LIN {X 0.039,Y -218.237,Z 1468.192,A 0.000,B 0.000,C 90.000,E1 34.612} C_DIS
LIN {X 0.042,Y -211.829,Z 1468.171,A 0.000,B 0.000,C 90.000,E1 30.718} C_DIS
LIN {X -0.038,Y -206.290,Z 1468.149,A 0.000,B 0.000,C 90.000,E1 26.796} C_DIS
LIN {X 0.085,Y -201.468,Z 1468.127,A 0.000,B 0.000,C 90.000,E1 22.770} C_DIS
LIN {X 0.019,Y -196.661,Z 1468.100,A 0.000,B 0.000,C 90.000,E1 17.946} C_DIS
LIN {X -0.013,Y -192.947,Z 1468.073,A 0.000,B 0.000,C 90.000,E1 13.063} C_DIS
LIN {X 0.033,Y -189.936,Z 1468.041,A 0.000,B 0.000,C 90.000,E1 7.296} C_DIS
LIN {X 0.003,Y -188.141,Z 1468.004,A 0.000,B 0.000,C 90.000,E1 0.688} C_DIS
LIN {X -0.094,Y -187.890,Z 1467.974,A 0.000,B 0.000,C 90.000,E1 355.412} C_DIS
LIN {X -0.024,Y -189.029,Z 1467.938,A 0.000,B 0.000,C 90.000,E1 348.757} C_DIS
LIN {X 0.018,Y -191.542,Z 1467.905,A 0.000,B 0.000,C 90.000,E1 342.960} C_DIS
LIN {X 0.031,Y -194.968,Z 1467.878,A 0.000,B 0.000,C 90.000,E1 338.028} C_DIS
LIN {X 0.048,Y -198.751,Z 1467.855,A 0.000,B 0.000,C 90.000,E1 333.948} C_DIS
LIN {X 0.000,Y -203.644,Z 1467.833,A 0.000,B 0.000,C 90.000,E1 329.921} C_DIS
LIN {X 0.050,Y -208.477,Z 1467.815,A 0.000,B 0.000,C 90.000,E1 326.707} C_DIS
LIN {X 0.045,Y -214.140,Z 1467.797,A 0.000,B 0.000,C 90.000,E1 323.543} C_DIS
LIN {X -0.033,Y -220.739,Z 1467.780,A 0.000,B 0.000,C 90.000,E1 320.436} C_DIS
LIN {X -0.092,Y -229.220,Z 1467.761,A 0.000,B 0.000,C 90.000,E1 316.986} C_DIS
LIN {X 0.104,Y -238.990,Z 1467.742,A 0.000,B 0.000,C 90.000,E1 313.542} C_DIS
LIN {X -0.060,Y -248.706,Z 1467.726,A 0.000,B 0.000,C 90.000,E1 310.620} C_DIS
LIN {X 0.027,Y -256.867,Z 1467.714,A 0.000,B 0.000,C 90.000,E1 308.418} C_DIS
LIN {X -0.032,Y -267.355,Z 1467.700,A 0.000,B 0.000,C 90.000,E1 305.931} C_DIS
LIN {X -0.147,Y -275.740,Z 1467.690,A 0.000,B 0.000,C 90.000,E1 304.199} C_DIS
LIN {X 0.156,Y -283.214,Z 1467.682,A 0.000,B 0.000,C 90.000,E1 302.752} C_DIS
LIN {X -0.016,Y -295.382,Z 1467.671,A 0.000,B 0.000,C 90.000,E1 300.747} C_DIS
LIN {X -0.006,Y -304.284,Z 1467.663,A 0.000,B 0.000,C 90.000,E1 299.411} C_DIS
LIN {X -0.072,Y -311.630,Z 1467.658,A 0.000,B 0.000,C 90.000,E1 298.437} C_DIS
LIN {X 0.129,Y -322.365,Z 1467.651,A 0.000,B 0.000,C 90.000,E1 297.129} C_DIS
LIN {X -0.024,Y -344.394,Z 1467.638,A 0.000,B 0.000,C 90.000,E1 294.823} C_DIS
LIN {X -0.093,Y -358.123,Z 1467.630,A 0.000,B 0.000,C 90.000,E1 293.462} C_DIS
LIN {X 0.175,Y -368.842,Z 1467.624,A 0.000,B 0.000,C 90.000,E1 292.333} C_DIS
LIN {X -0.167,Y -379.420,Z 1467.618,A 0.000,B 0.000,C 90.000,E1 291.280} C_DIS
LIN {X -0.060,Y -392.204,Z 1467.610,A 0.000,B 0.000,C 90.000,E1 289.885} C_DIS
LIN {X -0.036,Y -402.044,Z 1467.604,A 0.000,B 0.000,C 90.000,E1 288.779} C_DIS
LIN {X 0.133,Y -411.649,Z 1467.598,A 0.000,B 0.000,C 90.000,E1 287.638} C_DIS
LIN {X -0.221,Y -418.371,Z 1467.594,A 0.000,B 0.000,C 90.000,E1 286.858} C_DIS
LIN {X -0.109,Y -424.471,Z 1467.589,A 0.000,B 0.000,C 90.000,E1 286.024} C_DIS
LIN {X 0.057,Y -429.836,Z 1467.584,A 0.000,B 0.000,C 90.000,E1 285.190} C_DIS
LIN {X -0.142,Y -434.291,Z 1467.580,A 0.000,B 0.000,C 90.000,E1 284.411} C_DIS
LIN {X 0.007,Y -437.919,Z 1467.576,A 0.000,B 0.000,C 90.000,E1 283.592} C_DIS
LIN {X -0.013,Y -439.960,Z 1467.573,A 0.000,B 0.000,C 90.000,E1 283.063} C_DIS
LIN {X -0.024,Y -441.707,Z 1467.570,A 0.000,B 0.000,C 90.000,E1 282.535} C_DIS
LIN {X -0.024,Y -443.041,Z 1467.567,A 0.000,B 0.000,C 90.000,E1 282.007} C_DIS
LIN {X -0.013,Y -443.945,Z 1467.564,A 0.000,B 0.000,C 90.000,E1 281.478} C_DIS
LIN {X 0.003,Y -444.436,Z 1467.561,A 0.000,B 0.000,C 90.000,E1 280.950} C_DIS
LIN {X -0.058,Y -444.419,Z 1467.558,A 0.000,B 0.000,C 90.000,E1 280.433} C_DIS
LIN {X -0.035,Y -443.900,Z 1467.555,A 0.000,B 0.000,C 90.000,E1 279.905} C_DIS
LIN {X -0.014,Y -442.814,Z 1467.552,A 0.000,B 0.000,C 90.000,E1 279.378} C_DIS
LIN {X -0.069,Y -441.120,Z 1467.549,A 0.000,B 0.000,C 90.000,E1 278.859} C_DIS
LIN {X -0.126,Y -438.735,Z 1467.546,A 0.000,B 0.000,C 90.000,E1 278.341} C_DIS
LIN {X 0.086,Y -437.235,Z 1467.545,A 0.000,B 0.000,C 90.000,E1 278.049} C_DIS
LIN {X 0.005,Y -433.513,Z 1467.542,A 0.000,B 0.000,C 90.000,E1 277.530} C_DIS
LIN {X -0.038,Y -428.671,Z 1467.539,A 0.000,B 0.000,C 90.000,E1 277.004} C_DIS
LIN {X 0.024,Y -422.891,Z 1467.536,A 0.000,B 0.000,C 90.000,E1 276.486} C_DIS
LIN {X 0.018,Y -416.688,Z 1467.534,A 0.000,B 0.000,C 90.000,E1 276.030} C_DIS
LIN {X 0.045,Y -410.270,Z 1467.531,A 0.000,B 0.000,C 90.000,E1 275.625} C_DIS
LIN {X 0.086,Y -400.286,Z 1467.528,A 0.000,B 0.000,C 90.000,E1 275.106} C_DIS
LIN {X -0.114,Y -390.563,Z 1467.526,A 0.000,B 0.000,C 90.000,E1 274.702} C_DIS
LIN {X -0.087,Y -377.552,Z 1467.523,A 0.000,B 0.000,C 90.000,E1 274.188} C_DIS
LIN {X 0.178,Y -361.993,Z 1467.520,A 0.000,B 0.000,C 90.000,E1 273.555} C_DIS
LIN {X -0.158,Y -351.986,Z 1467.518,A 0.000,B 0.000,C 90.000,E1 273.269} C_DIS
LIN {X 0.128,Y -341.609,Z 1467.516,A 0.000,B 0.000,C 90.000,E1 272.922} C_DIS
LIN {X 0.001,Y -331.098,Z 1467.515,A 0.000,B 0.000,C 90.000,E1 272.694} C_DIS
LIN {X 0.066,Y -316.001,Z 1467.513,A 0.000,B 0.000,C 90.000,E1 272.407} C_DIS
LIN {X 0.068,Y -306.781,Z 1467.513,A 0.000,B 0.000,C 90.000,E1 272.293} C_DIS
LIN {X -0.016,Y -296.103,Z 1467.512,A 0.000,B 0.000,C 90.000,E1 272.236} C_DIS
LIN {X -0.068,Y -290.662,Z 1467.512,A 0.000,B 0.000,C 90.000,E1 272.236} C_DIS
LIN {X -0.075,Y -181.228,Z 1467.512,A 0.000,B 0.000,C 90.000,E1 272.236} C_DIS
LIN {X 0.089,Y -181.567,Z 1467.503,A 0.000,B 0.000,C 90.000,E1 270.458} C_DIS
LIN {X 0.078,Y -181.118,Z 1467.489,A 0.000,B 0.000,C 90.000,E1 267.936} C_DIS
LIN {X 0.066,Y -180.906,Z 1467.475,A 0.000,B 0.000,C 90.000,E1 265.412} C_DIS
LIN {X -0.058,Y -180.720,Z 1467.470,A 0.000,B 0.000,C 90.000,E1 264.609} C_DIS
LIN {X 0.040,Y -178.808,Z 1467.442,A 0.000,B 0.000,C 90.000,E1 259.511} C_DIS
LIN {X -0.052,Y -175.852,Z 1467.413,A 0.000,B 0.000,C 90.000,E1 254.448} C_DIS
LIN {X -0.071,Y -173.179,Z 1467.395,A 0.000,B 0.000,C 90.000,E1 251.040} C_DIS
LIN {X -0.068,Y -171.480,Z 1467.380,A 0.000,B 0.000,C 90.000,E1 248.465} C_DIS
LIN {X -0.080,Y -167.710,Z 1467.356,A 0.000,B 0.000,C 90.000,E1 244.152} C_DIS
LIN {X -0.063,Y -166.399,Z 1467.347,A 0.000,B 0.000,C 90.000,E1 242.410} C_DIS
LIN {X 0.075,Y -163.124,Z 1467.327,A 0.000,B 0.000,C 90.000,E1 238.869} C_DIS
LIN {X -0.099,Y -161.075,Z 1467.313,A 0.000,B 0.000,C 90.000,E1 236.294} C_DIS
LIN {X 0.012,Y -157.807,Z 1467.293,A 0.000,B 0.000,C 90.000,E1 232.718} C_DIS
LIN {X -0.050,Y -155.842,Z 1467.278,A 0.000,B 0.000,C 90.000,E1 230.070} C_DIS
LIN {X 0.006,Y -152.092,Z 1467.253,A 0.000,B 0.000,C 90.000,E1 225.567} C_DIS
LIN {X 0.025,Y -150.342,Z 1467.238,A 0.000,B 0.000,C 90.000,E1 222.852} C_DIS
LIN {X 0.046,Y -147.081,Z 1467.213,A 0.000,B 0.000,C 90.000,E1 218.302} C_DIS
LIN {X -0.051,Y -145.653,Z 1467.198,A 0.000,B 0.000,C 90.000,E1 215.598} C_DIS
LIN {X -0.046,Y -143.036,Z 1467.172,A 0.000,B 0.000,C 90.000,E1 211.003} C_DIS
LIN {X 0.080,Y -141.661,Z 1467.152,A 0.000,B 0.000,C 90.000,E1 207.257} C_DIS
LIN {X -0.001,Y -139.448,Z 1467.115,A 0.000,B 0.000,C 90.000,E1 200.791} C_DIS
LIN {X 0.052,Y -139.181,Z 1467.105,A 0.000,B 0.000,C 90.000,E1 198.906} C_DIS
LIN {X -0.057,Y -138.321,Z 1467.053,A 0.000,B 0.000,C 90.000,E1 189.613} C_DIS
LIN {X -0.050,Y -139.465,Z 1467.007,A 0.000,B 0.000,C 90.000,E1 181.203} C_DIS
LIN {X 0.030,Y -141.025,Z 1466.976,A 0.000,B 0.000,C 90.000,E1 175.584} C_DIS
LIN {X -0.015,Y -142.391,Z 1466.960,A 0.000,B 0.000,C 90.000,E1 172.818} C_DIS
LIN {X 0.048,Y -144.622,Z 1466.934,A 0.000,B 0.000,C 90.000,E1 168.173} C_DIS
LIN {X -0.033,Y -147.818,Z 1466.909,A 0.000,B 0.000,C 90.000,E1 163.614} C_DIS
LIN {X 0.053,Y -150.507,Z 1466.889,A 0.000,B 0.000,C 90.000,E1 159.934} C_DIS
LIN {X -0.067,Y -153.967,Z 1466.869,A 0.000,B 0.000,C 90.000,E1 156.357} C_DIS
LIN {X -0.005,Y -157.379,Z 1466.849,A 0.000,B 0.000,C 90.000,E1 152.743} C_DIS
LIN {X -0.063,Y -161.581,Z 1466.829,A 0.000,B 0.000,C 90.000,E1 149.203} C_DIS
LIN {X -0.052,Y -165.778,Z 1466.809,A 0.000,B 0.000,C 90.000,E1 145.674} C_DIS
LIN {X -0.065,Y -170.738,Z 1466.790,A 0.000,B 0.000,C 90.000,E1 142.190} C_DIS
LIN {X 0.092,Y -175.611,Z 1466.771,A 0.000,B 0.000,C 90.000,E1 138.690} C_DIS
LIN {X -0.037,Y -181.226,Z 1466.752,A 0.000,B 0.000,C 90.000,E1 135.324} C_DIS
LIN {X 0.093,Y -186.694,Z 1466.733,A 0.000,B 0.000,C 90.000,E1 131.919} C_DIS
LIN {X 0.045,Y -191.295,Z 1466.719,A 0.000,B 0.000,C 90.000,E1 129.439} C_DIS
LIN {X -0.023,Y -197.122,Z 1466.701,A 0.000,B 0.000,C 90.000,E1 126.171} C_DIS
LIN {X 0.020,Y -201.012,Z 1466.690,A 0.000,B 0.000,C 90.000,E1 124.199} C_DIS
LIN {X -0.005,Y -313.705,Z 1466.690,A 0.000,B 0.000,C 90.000,E1 124.199} C_DIS
LIN {X -0.163,Y -315.308,Z 1466.690,A 0.000,B 0.000,C 90.000,E1 124.199} C_DIS
LIN {X 0.195,Y -319.977,Z 1466.689,A 0.000,B 0.000,C 90.000,E1 123.913} C_DIS
LIN {X 0.113,Y -322.560,Z 1466.687,A 0.000,B 0.000,C 90.000,E1 123.706} C_DIS
LIN {X -0.075,Y -326.334,Z 1466.685,A 0.000,B 0.000,C 90.000,E1 123.245} C_DIS
LIN {X 0.018,Y -328.019,Z 1466.683,A 0.000,B 0.000,C 90.000,E1 122.911} C_DIS
LIN {X -0.057,Y -330.466,Z 1466.679,A 0.000,B 0.000,C 90.000,E1 122.291} C_DIS
LIN {X 0.069,Y -341.375,Z 1466.664,A 0.000,B 0.000,C 90.000,E1 119.461} C_DIS
LIN {X -0.168,Y -353.655,Z 1466.648,A 0.000,B 0.000,C 90.000,E1 116.744} C_DIS
LIN {X -0.052,Y -367.420,Z 1466.633,A 0.000,B 0.000,C 90.000,E1 114.027} C_DIS
LIN {X 0.054,Y -380.993,Z 1466.620,A 0.000,B 0.000,C 90.000,E1 111.663} C_DIS
LIN {X -0.142,Y -395.924,Z 1466.608,A 0.000,B 0.000,C 90.000,E1 109.396} C_DIS
LIN {X -0.119,Y -412.316,Z 1466.595,A 0.000,B 0.000,C 90.000,E1 107.149} C_DIS
LIN {X -0.056,Y -430.284,Z 1466.583,A 0.000,B 0.000,C 90.000,E1 104.954} C_DIS
LIN {X 0.052,Y -449.801,Z 1466.571,A 0.000,B 0.000,C 90.000,E1 102.827} C_DIS
LIN {X -0.114,Y -470.040,Z 1466.560,A 0.000,B 0.000,C 90.000,E1 100.894} C_DIS
LIN {X -0.163,Y -488.135,Z 1466.552,A 0.000,B 0.000,C 90.000,E1 99.321} C_DIS
LIN {X -0.088,Y -490.219,Z 1466.550,A 0.000,B 0.000,C 90.000,E1 99.095} C_DIS
LIN {X -0.188,Y -491.996,Z 1466.549,A 0.000,B 0.000,C 90.000,E1 98.859} C_DIS
LIN {X 0.198,Y -493.325,Z 1466.548,A 0.000,B 0.000,C 90.000,E1 98.568} C_DIS
LIN {X -0.058,Y -494.970,Z 1466.545,A 0.000,B 0.000,C 90.000,E1 98.106} C_DIS
LIN {X 0.186,Y -495.527,Z 1466.542,A 0.000,B 0.000,C 90.000,E1 97.587} C_DIS
LIN {X -0.051,Y -495.093,Z 1466.540,A 0.000,B 0.000,C 90.000,E1 97.125} C_DIS
LIN {X 0.206,Y -493.599,Z 1466.537,A 0.000,B 0.000,C 90.000,E1 96.606} C_DIS
LIN {X 0.116,Y -492.376,Z 1466.536,A 0.000,B 0.000,C 90.000,E1 96.372} C_DIS
LIN {X -0.040,Y -479.223,Z 1466.525,A 0.000,B 0.000,C 90.000,E1 94.416} C_DIS
LIN {X -0.115,Y -470.140,Z 1466.516,A 0.000,B 0.000,C 90.000,E1 92.922} C_DIS
LIN {X 0.033,Y -463.742,Z 1466.510,A 0.000,B 0.000,C 90.000,E1 91.892} C_DIS
LIN {X 0.128,Y -453.624,Z 1466.502,A 0.000,B 0.000,C 90.000,E1 90.344} C_DIS
LIN {X 0.163,Y -438.329,Z 1466.489,A 0.000,B 0.000,C 90.000,E1 87.993} C_DIS
LIN {X -0.171,Y -428.170,Z 1466.480,A 0.000,B 0.000,C 90.000,E1 86.445} C_DIS
LIN {X 0.007,Y -414.601,Z 1466.468,A 0.000,B 0.000,C 90.000,E1 84.261} C_DIS
LIN {X 0.154,Y -404.353,Z 1466.459,A 0.000,B 0.000,C 90.000,E1 82.591} C_DIS
LIN {X -0.092,Y -390.495,Z 1466.447,A 0.000,B 0.000,C 90.000,E1 80.387} C_DIS
LIN {X -0.094,Y -373.602,Z 1466.431,A 0.000,B 0.000,C 90.000,E1 77.521} C_DIS
LIN {X -0.033,Y -359.028,Z 1466.416,A 0.000,B 0.000,C 90.000,E1 74.866} C_DIS
LIN {X -0.122,Y -347.674,Z 1466.404,A 0.000,B 0.000,C 90.000,E1 72.779} C_DIS
LIN {X -0.039,Y -334.716,Z 1466.391,A 0.000,B 0.000,C 90.000,E1 70.315} C_DIS
LIN {X 0.057,Y -322.144,Z 1466.377,A 0.000,B 0.000,C 90.000,E1 67.794} C_DIS
LIN {X 0.051,Y -307.362,Z 1466.359,A 0.000,B 0.000,C 90.000,E1 64.588} C_DIS
LIN {X 0.002,Y -293.598,Z 1466.341,A 0.000,B 0.000,C 90.000,E1 61.307} C_DIS
LIN {X 0.102,Y -280.859,Z 1466.322,A 0.000,B 0.000,C 90.000,E1 57.916} C_DIS
LIN {X 0.002,Y -271.142,Z 1466.307,A 0.000,B 0.000,C 90.000,E1 55.182} C_DIS
LIN {X -0.032,Y -260.680,Z 1466.289,A 0.000,B 0.000,C 90.000,E1 52.029} C_DIS
LIN {X 0.135,Y -250.895,Z 1466.271,A 0.000,B 0.000,C 90.000,E1 48.771} C_DIS
LIN {X -0.023,Y -240.938,Z 1466.251,A 0.000,B 0.000,C 90.000,E1 45.162} C_DIS
LIN {X 0.022,Y -231.955,Z 1466.230,A 0.000,B 0.000,C 90.000,E1 41.434} C_DIS
LIN {X 0.021,Y -224.025,Z 1466.209,A 0.000,B 0.000,C 90.000,E1 37.649} C_DIS
LIN {X 0.086,Y -217.027,Z 1466.188,A 0.000,B 0.000,C 90.000,E1 33.785} C_DIS
LIN {X -0.061,Y -210.798,Z 1466.166,A 0.000,B 0.000,C 90.000,E1 29.922} C_DIS
LIN {X -0.082,Y -205.419,Z 1466.144,A 0.000,B 0.000,C 90.000,E1 25.976} C_DIS
LIN {X -0.060,Y -200.762,Z 1466.122,A 0.000,B 0.000,C 90.000,E1 21.972} C_DIS
LIN {X 0.036,Y -196.162,Z 1466.095,A 0.000,B 0.000,C 90.000,E1 17.094} C_DIS
LIN {X 0.072,Y -192.659,Z 1466.068,A 0.000,B 0.000,C 90.000,E1 12.187} C_DIS
LIN {X 0.004,Y -189.592,Z 1466.031,A 0.000,B 0.000,C 90.000,E1 5.625} C_DIS
LIN {X -0.034,Y -188.285,Z 1465.997,A 0.000,B 0.000,C 90.000,E1 359.542} C_DIS
LIN {X -0.047,Y -188.256,Z 1465.965,A 0.000,B 0.000,C 90.000,E1 353.742} C_DIS
LIN {X -0.028,Y -189.513,Z 1465.933,A 0.000,B 0.000,C 90.000,E1 347.937} C_DIS
LIN {X 0.083,Y -192.235,Z 1465.901,A 0.000,B 0.000,C 90.000,E1 342.127} C_DIS
LIN {X 0.004,Y -195.817,Z 1465.874,A 0.000,B 0.000,C 90.000,E1 337.230} C_DIS
LIN {X -0.054,Y -199.777,Z 1465.851,A 0.000,B 0.000,C 90.000,E1 333.179} C_DIS
LIN {X 0.027,Y -204.898,Z 1465.828,A 0.000,B 0.000,C 90.000,E1 329.125} C_DIS
LIN {X 0.047,Y -209.946,Z 1465.811,A 0.000,B 0.000,C 90.000,E1 325.928} C_DIS
LIN {X 0.083,Y -215.832,Z 1465.793,A 0.000,B 0.000,C 90.000,E1 322.763} C_DIS
LIN {X 0.014,Y -222.679,Z 1465.776,A 0.000,B 0.000,C 90.000,E1 319.666} C_DIS
LIN {X -0.084,Y -230.393,Z 1465.759,A 0.000,B 0.000,C 90.000,E1 316.620} C_DIS
LIN {X -0.020,Y -240.294,Z 1465.740,A 0.000,B 0.000,C 90.000,E1 313.218} C_DIS
LIN {X 0.032,Y -250.183,Z 1465.724,A 0.000,B 0.000,C 90.000,E1 310.253} C_DIS
LIN {X -0.018,Y -259.927,Z 1465.710,A 0.000,B 0.000,C 90.000,E1 307.729} C_DIS
LIN {X -0.029,Y -269.118,Z 1465.698,A 0.000,B 0.000,C 90.000,E1 305.598} C_DIS
LIN {X 0.048,Y -277.640,Z 1465.688,A 0.000,B 0.000,C 90.000,E1 303.833} C_DIS
LIN {X -0.087,Y -289.218,Z 1465.677,A 0.000,B 0.000,C 90.000,E1 301.799} C_DIS
LIN {X 0.094,Y -299.751,Z 1465.667,A 0.000,B 0.000,C 90.000,E1 300.079} C_DIS
LIN {X 0.163,Y -309.133,Z 1465.660,A 0.000,B 0.000,C 90.000,E1 298.743} C_DIS
LIN {X 0.171,Y -316.913,Z 1465.654,A 0.000,B 0.000,C 90.000,E1 297.769} C_DIS
LIN {X -0.167,Y -341.562,Z 1465.640,A 0.000,B 0.000,C 90.000,E1 295.155} C_DIS
LIN {X 0.059,Y -358.065,Z 1465.630,A 0.000,B 0.000,C 90.000,E1 293.462} C_DIS
LIN {X -0.007,Y -368.787,Z 1465.624,A 0.000,B 0.000,C 90.000,E1 292.386} C_DIS
LIN {X 0.027,Y -379.306,Z 1465.618,A 0.000,B 0.000,C 90.000,E1 291.280} C_DIS
LIN {X 0.033,Y -389.615,Z 1465.612,A 0.000,B 0.000,C 90.000,E1 290.174} C_DIS
LIN {X -0.162,Y -399.658,Z 1465.606,A 0.000,B 0.000,C 90.000,E1 289.087} C_DIS
LIN {X 0.048,Y -409.329,Z 1465.600,A 0.000,B 0.000,C 90.000,E1 287.946} C_DIS
LIN {X 0.203,Y -416.258,Z 1465.595,A 0.000,B 0.000,C 90.000,E1 287.094} C_DIS
LIN {X -0.112,Y -422.625,Z 1465.591,A 0.000,B 0.000,C 90.000,E1 286.315} C_DIS
LIN {X 0.038,Y -428.286,Z 1465.586,A 0.000,B 0.000,C 90.000,E1 285.481} C_DIS
LIN {X -0.045,Y -431.599,Z 1465.583,A 0.000,B 0.000,C 90.000,E1 284.954} C_DIS
LIN {X 0.187,Y -435.772,Z 1465.579,A 0.000,B 0.000,C 90.000,E1 284.120} C_DIS
LIN {X 0.155,Y -438.131,Z 1465.576,A 0.000,B 0.000,C 90.000,E1 283.592} C_DIS
LIN {X 0.138,Y -440.159,Z 1465.573,A 0.000,B 0.000,C 90.000,E1 283.063} C_DIS
LIN {X 0.128,Y -441.908,Z 1465.570,A 0.000,B 0.000,C 90.000,E1 282.535} C_DIS
LIN {X 0.130,Y -443.324,Z 1465.567,A 0.000,B 0.000,C 90.000,E1 282.007} C_DIS
LIN {X 0.142,Y -444.213,Z 1465.564,A 0.000,B 0.000,C 90.000,E1 281.478} C_DIS
LIN {X 0.160,Y -444.747,Z 1465.561,A 0.000,B 0.000,C 90.000,E1 280.950} C_DIS
LIN {X 0.100,Y -444.791,Z 1465.558,A 0.000,B 0.000,C 90.000,E1 280.433} C_DIS
LIN {X 0.125,Y -444.292,Z 1465.555,A 0.000,B 0.000,C 90.000,E1 279.905} C_DIS
LIN {X 0.148,Y -443.275,Z 1465.552,A 0.000,B 0.000,C 90.000,E1 279.378} C_DIS
LIN {X 0.095,Y -441.640,Z 1465.549,A 0.000,B 0.000,C 90.000,E1 278.859} C_DIS
LIN {X 0.039,Y -439.351,Z 1465.546,A 0.000,B 0.000,C 90.000,E1 278.341} C_DIS
LIN {X 0.030,Y -436.207,Z 1465.543,A 0.000,B 0.000,C 90.000,E1 277.814} C_DIS
LIN {X -0.055,Y -432.055,Z 1465.541,A 0.000,B 0.000,C 90.000,E1 277.296} C_DIS
LIN {X -0.158,Y -426.696,Z 1465.537,A 0.000,B 0.000,C 90.000,E1 276.777} C_DIS
LIN {X 0.036,Y -420.616,Z 1465.535,A 0.000,B 0.000,C 90.000,E1 276.258} C_DIS
LIN {X -0.145,Y -414.383,Z 1465.532,A 0.000,B 0.000,C 90.000,E1 275.853} C_DIS
LIN {X -0.037,Y -407.702,Z 1465.530,A 0.000,B 0.000,C 90.000,E1 275.454} C_DIS
LIN {X -0.137,Y -397.895,Z 1465.528,A 0.000,B 0.000,C 90.000,E1 274.992} C_DIS
LIN {X 0.126,Y -388.024,Z 1465.525,A 0.000,B 0.000,C 90.000,E1 274.531} C_DIS
LIN {X -0.109,Y -369.137,Z 1465.521,A 0.000,B 0.000,C 90.000,E1 273.841} C_DIS
LIN {X -0.166,Y -356.289,Z 1465.519,A 0.000,B 0.000,C 90.000,E1 273.383} C_DIS
LIN {X -0.068,Y -349.638,Z 1465.517,A 0.000,B 0.000,C 90.000,E1 273.154} C_DIS
LIN {X 0.132,Y -335.511,Z 1465.515,A 0.000,B 0.000,C 90.000,E1 272.751} C_DIS
LIN {X 0.158,Y -324.427,Z 1465.514,A 0.000,B 0.000,C 90.000,E1 272.522} C_DIS
LIN {X 0.039,Y -312.156,Z 1465.513,A 0.000,B 0.000,C 90.000,E1 272.350} C_DIS
LIN {X 0.088,Y -300.899,Z 1465.513,A 0.000,B 0.000,C 90.000,E1 272.236} C_DIS
LIN {X -0.072,Y -290.419,Z 1465.512,A 0.000,B 0.000,C 90.000,E1 272.236} C_DIS
LIN {X -0.078,Y -181.229,Z 1465.512,A 0.000,B 0.000,C 90.000,E1 272.236} C_DIS
LIN {X 0.086,Y -181.567,Z 1465.503,A 0.000,B 0.000,C 90.000,E1 270.458} C_DIS
LIN {X 0.075,Y -181.118,Z 1465.489,A 0.000,B 0.000,C 90.000,E1 267.936} C_DIS
LIN {X 0.063,Y -180.907,Z 1465.475,A 0.000,B 0.000,C 90.000,E1 265.412} C_DIS
LIN {X -0.061,Y -180.719,Z 1465.470,A 0.000,B 0.000,C 90.000,E1 264.609} C_DIS
LIN {X 0.037,Y -178.807,Z 1465.442,A 0.000,B 0.000,C 90.000,E1 259.511} C_DIS
LIN {X -0.056,Y -175.852,Z 1465.413,A 0.000,B 0.000,C 90.000,E1 254.448} C_DIS
LIN {X -0.073,Y -173.178,Z 1465.395,A 0.000,B 0.000,C 90.000,E1 251.040} C_DIS
LIN {X -0.071,Y -171.479,Z 1465.380,A 0.000,B 0.000,C 90.000,E1 248.465} C_DIS
LIN {X -0.083,Y -167.710,Z 1465.356,A 0.000,B 0.000,C 90.000,E1 244.152} C_DIS
LIN {X 0.080,Y -166.398,Z 1465.347,A 0.000,B 0.000,C 90.000,E1 242.359} C_DIS
LIN {X 0.072,Y -163.123,Z 1465.327,A 0.000,B 0.000,C 90.000,E1 238.869} C_DIS
LIN {X -0.101,Y -161.073,Z 1465.313,A 0.000,B 0.000,C 90.000,E1 236.294} C_DIS
LIN {X 0.008,Y -157.806,Z 1465.293,A 0.000,B 0.000,C 90.000,E1 232.718} C_DIS
LIN {X -0.053,Y -155.841,Z 1465.278,A 0.000,B 0.000,C 90.000,E1 230.070} C_DIS
LIN {X 0.003,Y -152.092,Z 1465.253,A 0.000,B 0.000,C 90.000,E1 225.567} C_DIS
LIN {X 0.022,Y -150.342,Z 1465.238,A 0.000,B 0.000,C 90.000,E1 222.852} C_DIS
LIN {X 0.043,Y -147.081,Z 1465.213,A 0.000,B 0.000,C 90.000,E1 218.302} C_DIS
LIN {X -0.054,Y -145.654,Z 1465.198,A 0.000,B 0.000,C 90.000,E1 215.598} C_DIS
LIN {X -0.049,Y -143.036,Z 1465.172,A 0.000,B 0.000,C 90.000,E1 211.003} C_DIS
LIN {X 0.077,Y -141.660,Z 1465.152,A 0.000,B 0.000,C 90.000,E1 207.257} C_DIS
LIN {X -0.004,Y -139.448,Z 1465.115,A 0.000,B 0.000,C 90.000,E1 200.791} C_DIS
LIN {X 0.048,Y -139.181,Z 1465.105,A 0.000,B 0.000,C 90.000,E1 198.906} C_DIS
LIN {X -0.059,Y -138.320,Z 1465.053,A 0.000,B 0.000,C 90.000,E1 189.613} C_DIS
LIN {X -0.053,Y -139.465,Z 1465.007,A 0.000,B 0.000,C 90.000,E1 181.203} C_DIS
LIN {X 0.027,Y -141.027,Z 1464.976,A 0.000,B 0.000,C 90.000,E1 175.584} C_DIS
LIN {X -0.018,Y -142.391,Z 1464.960,A 0.000,B 0.000,C 90.000,E1 172.818} C_DIS
LIN {X 0.045,Y -144.623,Z 1464.934,A 0.000,B 0.000,C 90.000,E1 168.173} C_DIS
LIN {X -0.036,Y -147.817,Z 1464.909,A 0.000,B 0.000,C 90.000,E1 163.614} C_DIS
LIN {X 0.051,Y -150.508,Z 1464.889,A 0.000,B 0.000,C 90.000,E1 159.934} C_DIS
LIN {X -0.070,Y -153.968,Z 1464.869,A 0.000,B 0.000,C 90.000,E1 156.357} C_DIS
LIN {X -0.008,Y -157.380,Z 1464.849,A 0.000,B 0.000,C 90.000,E1 152.743} C_DIS
LIN {X -0.066,Y -161.583,Z 1464.829,A 0.000,B 0.000,C 90.000,E1 149.203} C_DIS
LIN {X -0.055,Y -165.779,Z 1464.809,A 0.000,B 0.000,C 90.000,E1 145.674} C_DIS
LIN {X -0.069,Y -170.740,Z 1464.790,A 0.000,B 0.000,C 90.000,E1 142.190} C_DIS
LIN {X 0.089,Y -175.612,Z 1464.771,A 0.000,B 0.000,C 90.000,E1 138.690} C_DIS
LIN {X -0.041,Y -181.228,Z 1464.752,A 0.000,B 0.000,C 90.000,E1 135.324} C_DIS
LIN {X 0.090,Y -186.696,Z 1464.733,A 0.000,B 0.000,C 90.000,E1 131.919} C_DIS
LIN {X 0.042,Y -191.297,Z 1464.719,A 0.000,B 0.000,C 90.000,E1 129.439} C_DIS
LIN {X -0.026,Y -197.125,Z 1464.701,A 0.000,B 0.000,C 90.000,E1 126.171} C_DIS
LIN {X -0.051,Y -200.966,Z 1464.690,A 0.000,B 0.000,C 90.000,E1 124.246} C_DIS
LIN {X 0.132,Y -313.639,Z 1464.690,A 0.000,B 0.000,C 90.000,E1 124.199} C_DIS
LIN {X -0.101,Y -319.853,Z 1464.689,A 0.000,B 0.000,C 90.000,E1 123.992} C_DIS
LIN {X 0.108,Y -322.706,Z 1464.687,A 0.000,B 0.000,C 90.000,E1 123.706} C_DIS
LIN {X 0.058,Y -326.421,Z 1464.685,A 0.000,B 0.000,C 90.000,E1 123.214} C_DIS
LIN {X 0.149,Y -328.062,Z 1464.683,A 0.000,B 0.000,C 90.000,E1 122.880} C_DIS
LIN {X -0.155,Y -332.785,Z 1464.676,A 0.000,B 0.000,C 90.000,E1 121.671} C_DIS
LIN {X 0.159,Y -343.994,Z 1464.660,A 0.000,B 0.000,C 90.000,E1 118.821} C_DIS
LIN {X 0.005,Y -356.598,Z 1464.645,A 0.000,B 0.000,C 90.000,E1 116.104} C_DIS
LIN {X 0.210,Y -370.711,Z 1464.630,A 0.000,B 0.000,C 90.000,E1 113.387} C_DIS
LIN {X -0.098,Y -384.619,Z 1464.617,A 0.000,B 0.000,C 90.000,E1 111.099} C_DIS
LIN {X 0.157,Y -399.909,Z 1464.604,A 0.000,B 0.000,C 90.000,E1 108.779} C_DIS
LIN {X 0.040,Y -416.688,Z 1464.592,A 0.000,B 0.000,C 90.000,E1 106.567} C_DIS
LIN {X -0.077,Y -435.076,Z 1464.580,A 0.000,B 0.000,C 90.000,E1 104.411} C_DIS
LIN {X 0.189,Y -454.850,Z 1464.568,A 0.000,B 0.000,C 90.000,E1 102.299} C_DIS
LIN {X -0.100,Y -475.226,Z 1464.558,A 0.000,B 0.000,C 90.000,E1 100.423} C_DIS
LIN {X -0.217,Y -488.167,Z 1464.552,A 0.000,B 0.000,C 90.000,E1 99.321} C_DIS
LIN {X -0.142,Y -490.215,Z 1464.550,A 0.000,B 0.000,C 90.000,E1 99.095} C_DIS
LIN {X -0.242,Y -491.965,Z 1464.549,A 0.000,B 0.000,C 90.000,E1 98.859} C_DIS
LIN {X 0.144,Y -493.274,Z 1464.548,A 0.000,B 0.000,C 90.000,E1 98.568} C_DIS
LIN {X -0.112,Y -494.888,Z 1464.545,A 0.000,B 0.000,C 90.000,E1 98.106} C_DIS
LIN {X 0.131,Y -495.421,Z 1464.542,A 0.000,B 0.000,C 90.000,E1 97.587} C_DIS
LIN {X -0.106,Y -494.961,Z 1464.540,A 0.000,B 0.000,C 90.000,E1 97.125} C_DIS
LIN {X 0.151,Y -493.439,Z 1464.537,A 0.000,B 0.000,C 90.000,E1 96.606} C_DIS
LIN {X 0.060,Y -492.198,Z 1464.535,A 0.000,B 0.000,C 90.000,E1 96.372} C_DIS
LIN {X -0.098,Y -479.013,Z 1464.524,A 0.000,B 0.000,C 90.000,E1 94.416} C_DIS
LIN {X -0.175,Y -469.920,Z 1464.516,A 0.000,B 0.000,C 90.000,E1 92.922} C_DIS
LIN {X -0.030,Y -463.521,Z 1464.510,A 0.000,B 0.000,C 90.000,E1 91.892} C_DIS
LIN {X 0.064,Y -453.397,Z 1464.502,A 0.000,B 0.000,C 90.000,E1 90.344} C_DIS
LIN {X -0.173,Y -436.468,Z 1464.487,A 0.000,B 0.000,C 90.000,E1 87.764} C_DIS
LIN {X 0.055,Y -424.631,Z 1464.477,A 0.000,B 0.000,C 90.000,E1 85.869} C_DIS
LIN {X 0.062,Y -412.806,Z 1464.467,A 0.000,B 0.000,C 90.000,E1 83.970} C_DIS
LIN {X 0.181,Y -402.524,Z 1464.457,A 0.000,B 0.000,C 90.000,E1 82.299} C_DIS
LIN {X -0.104,Y -388.740,Z 1464.445,A 0.000,B 0.000,C 90.000,E1 80.095} C_DIS
LIN {X 0.203,Y -373.565,Z 1464.431,A 0.000,B 0.000,C 90.000,E1 77.465} C_DIS
LIN {X -0.155,Y -360.622,Z 1464.417,A 0.000,B 0.000,C 90.000,E1 75.172} C_DIS
LIN {X -0.150,Y -350.909,Z 1464.407,A 0.000,B 0.000,C 90.000,E1 73.378} C_DIS
LIN {X 0.012,Y -339.507,Z 1464.396,A 0.000,B 0.000,C 90.000,E1 71.221} C_DIS
LIN {X 0.108,Y -326.794,Z 1464.382,A 0.000,B 0.000,C 90.000,E1 68.720} C_DIS
LIN {X 0.032,Y -310.200,Z 1464.362,A 0.000,B 0.000,C 90.000,E1 65.229} C_DIS
LIN {X -0.069,Y -296.181,Z 1464.344,A 0.000,B 0.000,C 90.000,E1 61.975} C_DIS
LIN {X -0.042,Y -283.265,Z 1464.326,A 0.000,B 0.000,C 90.000,E1 58.614} C_DIS
LIN {X -0.083,Y -273.483,Z 1464.310,A 0.000,B 0.000,C 90.000,E1 55.881} C_DIS
LIN {X 0.000,Y -262.926,Z 1464.293,A 0.000,B 0.000,C 90.000,E1 52.718} C_DIS
LIN {X -0.136,Y -253.019,Z 1464.275,A 0.000,B 0.000,C 90.000,E1 49.542} C_DIS
LIN {X -0.045,Y -242.938,Z 1464.255,A 0.000,B 0.000,C 90.000,E1 45.891} C_DIS
LIN {X 0.067,Y -233.815,Z 1464.234,A 0.000,B 0.000,C 90.000,E1 42.162} C_DIS
LIN {X 0.099,Y -225.705,Z 1464.213,A 0.000,B 0.000,C 90.000,E1 38.382} C_DIS
LIN {X 0.039,Y -218.569,Z 1464.192,A 0.000,B 0.000,C 90.000,E1 34.565} C_DIS
LIN {X 0.060,Y -212.151,Z 1464.171,A 0.000,B 0.000,C 90.000,E1 30.669} C_DIS
LIN {X -0.005,Y -206.611,Z 1464.149,A 0.000,B 0.000,C 90.000,E1 26.744} C_DIS
LIN {X -0.052,Y -201.819,Z 1464.126,A 0.000,B 0.000,C 90.000,E1 22.770} C_DIS
LIN {X -0.040,Y -197.057,Z 1464.099,A 0.000,B 0.000,C 90.000,E1 17.928} C_DIS
LIN {X 0.072,Y -193.423,Z 1464.072,A 0.000,B 0.000,C 90.000,E1 13.008} C_DIS
LIN {X -0.047,Y -190.477,Z 1464.040,A 0.000,B 0.000,C 90.000,E1 7.296} C_DIS
LIN {X 0.038,Y -188.837,Z 1464.008,A 0.000,B 0.000,C 90.000,E1 1.489} C_DIS
LIN {X -0.078,Y -188.398,Z 1463.974,A 0.000,B 0.000,C 90.000,E1 355.412} C_DIS
LIN {X 0.017,Y -189.478,Z 1463.938,A 0.000,B 0.000,C 90.000,E1 348.757} C_DIS
LIN {X 0.079,Y -191.936,Z 1463.906,A 0.000,B 0.000,C 90.000,E1 342.960} C_DIS
LIN {X 0.035,Y -195.281,Z 1463.878,A 0.000,B 0.000,C 90.000,E1 338.050} C_DIS
LIN {X 0.048,Y -199.036,Z 1463.855,A 0.000,B 0.000,C 90.000,E1 333.973} C_DIS
LIN {X -0.003,Y -203.931,Z 1463.833,A 0.000,B 0.000,C 90.000,E1 329.950} C_DIS
LIN {X -0.016,Y -208.732,Z 1463.815,A 0.000,B 0.000,C 90.000,E1 326.755} C_DIS
LIN {X 0.036,Y -214.425,Z 1463.798,A 0.000,B 0.000,C 90.000,E1 323.577} C_DIS
LIN {X 0.096,Y -221.026,Z 1463.780,A 0.000,B 0.000,C 90.000,E1 320.436} C_DIS
LIN {X 0.050,Y -229.511,Z 1463.761,A 0.000,B 0.000,C 90.000,E1 316.986} C_DIS
LIN {X -0.077,Y -239.289,Z 1463.742,A 0.000,B 0.000,C 90.000,E1 313.623} C_DIS
LIN {X 0.112,Y -249.036,Z 1463.726,A 0.000,B 0.000,C 90.000,E1 310.620} C_DIS
LIN {X 0.043,Y -258.627,Z 1463.712,A 0.000,B 0.000,C 90.000,E1 308.096} C_DIS
LIN {X 0.010,Y -267.675,Z 1463.700,A 0.000,B 0.000,C 90.000,E1 305.964} C_DIS
LIN {X 0.063,Y -275.988,Z 1463.690,A 0.000,B 0.000,C 90.000,E1 304.199} C_DIS
LIN {X -0.016,Y -283.350,Z 1463.682,A 0.000,B 0.000,C 90.000,E1 302.832} C_DIS
LIN {X -0.039,Y -295.477,Z 1463.671,A 0.000,B 0.000,C 90.000,E1 300.797} C_DIS
LIN {X -0.031,Y -304.364,Z 1463.664,A 0.000,B 0.000,C 90.000,E1 299.461} C_DIS
LIN {X -0.064,Y -314.264,Z 1463.656,A 0.000,B 0.000,C 90.000,E1 298.153} C_DIS
LIN {X -0.186,Y -327.935,Z 1463.648,A 0.000,B 0.000,C 90.000,E1 296.616} C_DIS
LIN {X 0.065,Y -350.047,Z 1463.635,A 0.000,B 0.000,C 90.000,E1 294.283} C_DIS
LIN {X 0.021,Y -363.413,Z 1463.628,A 0.000,B 0.000,C 90.000,E1 292.950} C_DIS
LIN {X 0.141,Y -373.989,Z 1463.621,A 0.000,B 0.000,C 90.000,E1 291.844} C_DIS
LIN {X 0.028,Y -386.947,Z 1463.614,A 0.000,B 0.000,C 90.000,E1 290.482} C_DIS
LIN {X 0.115,Y -394.607,Z 1463.609,A 0.000,B 0.000,C 90.000,E1 289.631} C_DIS
LIN {X 0.029,Y -407.049,Z 1463.601,A 0.000,B 0.000,C 90.000,E1 288.236} C_DIS
LIN {X -0.135,Y -416.392,Z 1463.595,A 0.000,B 0.000,C 90.000,E1 287.149} C_DIS
LIN {X -0.051,Y -422.793,Z 1463.591,A 0.000,B 0.000,C 90.000,E1 286.315} C_DIS
LIN {X 0.103,Y -428.486,Z 1463.586,A 0.000,B 0.000,C 90.000,E1 285.481} C_DIS
LIN {X 0.021,Y -431.826,Z 1463.583,A 0.000,B 0.000,C 90.000,E1 284.954} C_DIS
LIN {X -0.166,Y -436.013,Z 1463.579,A 0.000,B 0.000,C 90.000,E1 284.175} C_DIS
LIN {X 0.004,Y -439.417,Z 1463.574,A 0.000,B 0.000,C 90.000,E1 283.355} C_DIS
LIN {X 0.208,Y -442.166,Z 1463.570,A 0.000,B 0.000,C 90.000,E1 282.535} C_DIS
LIN {X 0.212,Y -443.540,Z 1463.567,A 0.000,B 0.000,C 90.000,E1 282.007} C_DIS
LIN {X 0.225,Y -444.515,Z 1463.564,A 0.000,B 0.000,C 90.000,E1 281.478} C_DIS
LIN {X 0.245,Y -445.051,Z 1463.561,A 0.000,B 0.000,C 90.000,E1 280.950} C_DIS
LIN {X 0.187,Y -445.132,Z 1463.558,A 0.000,B 0.000,C 90.000,E1 280.433} C_DIS
LIN {X 0.214,Y -444.669,Z 1463.555,A 0.000,B 0.000,C 90.000,E1 279.905} C_DIS
LIN {X 0.238,Y -443.719,Z 1463.552,A 0.000,B 0.000,C 90.000,E1 279.378} C_DIS
LIN {X 0.187,Y -442.134,Z 1463.549,A 0.000,B 0.000,C 90.000,E1 278.859} C_DIS
LIN {X 0.133,Y -439.878,Z 1463.546,A 0.000,B 0.000,C 90.000,E1 278.341} C_DIS
LIN {X 0.127,Y -436.828,Z 1463.543,A 0.000,B 0.000,C 90.000,E1 277.814} C_DIS
LIN {X 0.043,Y -432.751,Z 1463.541,A 0.000,B 0.000,C 90.000,E1 277.296} C_DIS
LIN {X -0.057,Y -427.490,Z 1463.538,A 0.000,B 0.000,C 90.000,E1 276.777} C_DIS
LIN {X 0.096,Y -421.398,Z 1463.535,A 0.000,B 0.000,C 90.000,E1 276.258} C_DIS
LIN {X -0.123,Y -415.118,Z 1463.532,A 0.000,B 0.000,C 90.000,E1 275.853} C_DIS
LIN {X -0.024,Y -408.522,Z 1463.530,A 0.000,B 0.000,C 90.000,E1 275.454} C_DIS
LIN {X -0.158,Y -398.622,Z 1463.528,A 0.000,B 0.000,C 90.000,E1 274.992} C_DIS
LIN {X 0.122,Y -388.831,Z 1463.525,A 0.000,B 0.000,C 90.000,E1 274.531} C_DIS
LIN {X -0.125,Y -369.832,Z 1463.521,A 0.000,B 0.000,C 90.000,E1 273.841} C_DIS
LIN {X -0.175,Y -357.026,Z 1463.519,A 0.000,B 0.000,C 90.000,E1 273.383} C_DIS
LIN {X -0.077,Y -350.398,Z 1463.517,A 0.000,B 0.000,C 90.000,E1 273.154} C_DIS
LIN {X -0.054,Y -339.740,Z 1463.516,A 0.000,B 0.000,C 90.000,E1 272.865} C_DIS
LIN {X -0.101,Y -329.040,Z 1463.515,A 0.000,B 0.000,C 90.000,E1 272.636} C_DIS
LIN {X 0.095,Y -317.771,Z 1463.513,A 0.000,B 0.000,C 90.000,E1 272.407} C_DIS
LIN {X 0.099,Y -308.487,Z 1463.513,A 0.000,B 0.000,C 90.000,E1 272.293} C_DIS
LIN {X 0.015,Y -298.734,Z 1463.512,A 0.000,B 0.000,C 90.000,E1 272.236} C_DIS
LIN {X -0.041,Y -295.301,Z 1463.512,A 0.000,B 0.000,C 90.000,E1 272.236} C_DIS
LIN {X -0.058,Y -181.228,Z 1463.512,A 0.000,B 0.000,C 90.000,E1 272.236} C_DIS
LIN {X -0.080,Y -181.567,Z 1463.503,A 0.000,B 0.000,C 90.000,E1 270.516} C_DIS
LIN {X 0.091,Y -181.119,Z 1463.489,A 0.000,B 0.000,C 90.000,E1 267.936} C_DIS
LIN {X 0.079,Y -180.906,Z 1463.475,A 0.000,B 0.000,C 90.000,E1 265.412} C_DIS
LIN {X -0.045,Y -180.722,Z 1463.470,A 0.000,B 0.000,C 90.000,E1 264.609} C_DIS
LIN {X 0.054,Y -178.809,Z 1463.442,A 0.000,B 0.000,C 90.000,E1 259.511} C_DIS
LIN {X -0.039,Y -175.855,Z 1463.414,A 0.000,B 0.000,C 90.000,E1 254.448} C_DIS
LIN {X -0.057,Y -173.182,Z 1463.395,A 0.000,B 0.000,C 90.000,E1 251.040} C_DIS
LIN {X -0.056,Y -171.483,Z 1463.380,A 0.000,B 0.000,C 90.000,E1 248.465} C_DIS
LIN {X -0.067,Y -167.713,Z 1463.356,A 0.000,B 0.000,C 90.000,E1 244.152} C_DIS
LIN {X -0.050,Y -166.404,Z 1463.347,A 0.000,B 0.000,C 90.000,E1 242.410} C_DIS
LIN {X 0.088,Y -163.128,Z 1463.327,A 0.000,B 0.000,C 90.000,E1 238.869} C_DIS
LIN {X -0.086,Y -161.080,Z 1463.313,A 0.000,B 0.000,C 90.000,E1 236.294} C_DIS
LIN {X 0.024,Y -157.810,Z 1463.293,A 0.000,B 0.000,C 90.000,E1 232.718} C_DIS
LIN {X -0.038,Y -155.845,Z 1463.278,A 0.000,B 0.000,C 90.000,E1 230.070} C_DIS
LIN {X 0.018,Y -152.096,Z 1463.253,A 0.000,B 0.000,C 90.000,E1 225.567} C_DIS
LIN {X 0.036,Y -150.346,Z 1463.238,A 0.000,B 0.000,C 90.000,E1 222.852} C_DIS
LIN {X 0.057,Y -147.083,Z 1463.213,A 0.000,B 0.000,C 90.000,E1 218.302} C_DIS
LIN {X -0.039,Y -145.656,Z 1463.198,A 0.000,B 0.000,C 90.000,E1 215.598} C_DIS
LIN {X -0.035,Y -143.039,Z 1463.172,A 0.000,B 0.000,C 90.000,E1 211.003} C_DIS
LIN {X -0.035,Y -141.663,Z 1463.152,A 0.000,B 0.000,C 90.000,E1 207.308} C_DIS
LIN {X 0.010,Y -139.449,Z 1463.115,A 0.000,B 0.000,C 90.000,E1 200.791} C_DIS
LIN {X 0.063,Y -139.182,Z 1463.105,A 0.000,B 0.000,C 90.000,E1 198.906} C_DIS
LIN {X -0.045,Y -138.321,Z 1463.053,A 0.000,B 0.000,C 90.000,E1 189.613} C_DIS
LIN {X -0.039,Y -139.463,Z 1463.007,A 0.000,B 0.000,C 90.000,E1 181.203} C_DIS
LIN {X 0.041,Y -141.024,Z 1462.976,A 0.000,B 0.000,C 90.000,E1 175.584} C_DIS
LIN {X -0.004,Y -142.389,Z 1462.960,A 0.000,B 0.000,C 90.000,E1 172.818} C_DIS
LIN {X 0.059,Y -144.620,Z 1462.934,A 0.000,B 0.000,C 90.000,E1 168.173} C_DIS
LIN {X -0.022,Y -147.814,Z 1462.909,A 0.000,B 0.000,C 90.000,E1 163.614} C_DIS
LIN {X 0.065,Y -150.504,Z 1462.889,A 0.000,B 0.000,C 90.000,E1 159.934} C_DIS
LIN {X -0.055,Y -153.963,Z 1462.869,A 0.000,B 0.000,C 90.000,E1 156.357} C_DIS
LIN {X 0.007,Y -157.374,Z 1462.849,A 0.000,B 0.000,C 90.000,E1 152.743} C_DIS
LIN {X -0.050,Y -161.576,Z 1462.829,A 0.000,B 0.000,C 90.000,E1 149.203} C_DIS
LIN {X -0.038,Y -165.773,Z 1462.809,A 0.000,B 0.000,C 90.000,E1 145.674} C_DIS
LIN {X -0.053,Y -170.731,Z 1462.790,A 0.000,B 0.000,C 90.000,E1 142.190} C_DIS
LIN {X -0.011,Y -175.604,Z 1462.771,A 0.000,B 0.000,C 90.000,E1 138.728} C_DIS
LIN {X -0.024,Y -181.220,Z 1462.752,A 0.000,B 0.000,C 90.000,E1 135.324} C_DIS
LIN {X -0.032,Y -186.686,Z 1462.733,A 0.000,B 0.000,C 90.000,E1 131.962} C_DIS
LIN {X 0.060,Y -191.288,Z 1462.719,A 0.000,B 0.000,C 90.000,E1 129.439} C_DIS
LIN {X -0.009,Y -197.114,Z 1462.701,A 0.000,B 0.000,C 90.000,E1 126.171} C_DIS
LIN {X -0.056,Y -200.912,Z 1462.690,A 0.000,B 0.000,C 90.000,E1 124.278} C_DIS
LIN {X 0.042,Y -313.072,Z 1462.690,A 0.000,B 0.000,C 90.000,E1 124.246} C_DIS
LIN {X 0.162,Y -314.792,Z 1462.690,A 0.000,B 0.000,C 90.000,E1 124.199} C_DIS
LIN {X -0.072,Y -320.032,Z 1462.689,A 0.000,B 0.000,C 90.000,E1 123.992} C_DIS
LIN {X 0.136,Y -322.791,Z 1462.687,A 0.000,B 0.000,C 90.000,E1 123.706} C_DIS
LIN {X 0.008,Y -326.507,Z 1462.685,A 0.000,B 0.000,C 90.000,E1 123.214} C_DIS
LIN {X 0.100,Y -328.104,Z 1462.683,A 0.000,B 0.000,C 90.000,E1 122.880} C_DIS
LIN {X -0.046,Y -342.695,Z 1462.662,A 0.000,B 0.000,C 90.000,E1 119.155} C_DIS
LIN {X -0.085,Y -355.145,Z 1462.647,A 0.000,B 0.000,C 90.000,E1 116.411} C_DIS
LIN {X 0.074,Y -369.087,Z 1462.632,A 0.000,B 0.000,C 90.000,E1 113.695} C_DIS
LIN {X 0.076,Y -382.831,Z 1462.619,A 0.000,B 0.000,C 90.000,E1 111.354} C_DIS
LIN {X -0.076,Y -397.948,Z 1462.606,A 0.000,B 0.000,C 90.000,E1 109.087} C_DIS
LIN {X -0.126,Y -414.541,Z 1462.594,A 0.000,B 0.000,C 90.000,E1 106.858} C_DIS
LIN {X 0.000,Y -432.725,Z 1462.581,A 0.000,B 0.000,C 90.000,E1 104.662} C_DIS
LIN {X -0.188,Y -452.375,Z 1462.570,A 0.000,B 0.000,C 90.000,E1 102.591} C_DIS
LIN {X -0.193,Y -472.686,Z 1462.559,A 0.000,B 0.000,C 90.000,E1 100.658} C_DIS
LIN {X 0.208,Y -488.199,Z 1462.552,A 0.000,B 0.000,C 90.000,E1 99.265} C_DIS
LIN {X -0.198,Y -490.211,Z 1462.550,A 0.000,B 0.000,C 90.000,E1 99.095} C_DIS
LIN {X 0.187,Y -491.932,Z 1462.549,A 0.000,B 0.000,C 90.000,E1 98.803} C_DIS
LIN {X 0.087,Y -493.221,Z 1462.548,A 0.000,B 0.000,C 90.000,E1 98.568} C_DIS
LIN {X -0.170,Y -494.803,Z 1462.545,A 0.000,B 0.000,C 90.000,E1 98.106} C_DIS
LIN {X 0.074,Y -495.309,Z 1462.542,A 0.000,B 0.000,C 90.000,E1 97.587} C_DIS
LIN {X -0.165,Y -494.824,Z 1462.539,A 0.000,B 0.000,C 90.000,E1 97.125} C_DIS
LIN {X 0.092,Y -493.271,Z 1462.537,A 0.000,B 0.000,C 90.000,E1 96.606} C_DIS
LIN {X 0.002,Y -492.010,Z 1462.535,A 0.000,B 0.000,C 90.000,E1 96.372} C_DIS
LIN {X -0.160,Y -478.804,Z 1462.524,A 0.000,B 0.000,C 90.000,E1 94.416} C_DIS
LIN {X 0.230,Y -469.711,Z 1462.516,A 0.000,B 0.000,C 90.000,E1 92.865} C_DIS
LIN {X -0.096,Y -463.298,Z 1462.510,A 0.000,B 0.000,C 90.000,E1 91.892} C_DIS
LIN {X -0.004,Y -453.163,Z 1462.502,A 0.000,B 0.000,C 90.000,E1 90.344} C_DIS
LIN {X 0.191,Y -436.263,Z 1462.487,A 0.000,B 0.000,C 90.000,E1 87.707} C_DIS
LIN {X -0.180,Y -426.157,Z 1462.479,A 0.000,B 0.000,C 90.000,E1 86.159} C_DIS
LIN {X -0.137,Y -414.398,Z 1462.468,A 0.000,B 0.000,C 90.000,E1 84.261} C_DIS
LIN {X 0.010,Y -404.200,Z 1462.459,A 0.000,B 0.000,C 90.000,E1 82.591} C_DIS
LIN {X 0.085,Y -392.124,Z 1462.448,A 0.000,B 0.000,C 90.000,E1 80.622} C_DIS
LIN {X 0.076,Y -378.529,Z 1462.435,A 0.000,B 0.000,C 90.000,E1 78.342} C_DIS
LIN {X 0.181,Y -363.797,Z 1462.421,A 0.000,B 0.000,C 90.000,E1 75.700} C_DIS
LIN {X 0.139,Y -354.132,Z 1462.411,A 0.000,B 0.000,C 90.000,E1 73.921} C_DIS
LIN {X 0.034,Y -342.738,Z 1462.399,A 0.000,B 0.000,C 90.000,E1 71.819} C_DIS
LIN {X 0.098,Y -329.908,Z 1462.385,A 0.000,B 0.000,C 90.000,E1 69.337} C_DIS
LIN {X -0.003,Y -313.058,Z 1462.366,A 0.000,B 0.000,C 90.000,E1 65.869} C_DIS
LIN {X -0.044,Y -300.223,Z 1462.350,A 0.000,B 0.000,C 90.000,E1 62.948} C_DIS
LIN {X -0.038,Y -286.977,Z 1462.331,A 0.000,B 0.000,C 90.000,E1 59.616} C_DIS
LIN {X -0.139,Y -277.059,Z 1462.316,A 0.000,B 0.000,C 90.000,E1 56.914} C_DIS
LIN {X -0.033,Y -265.177,Z 1462.297,A 0.000,B 0.000,C 90.000,E1 53.417} C_DIS
LIN {X 0.092,Y -255.130,Z 1462.279,A 0.000,B 0.000,C 90.000,E1 50.194} C_DIS
LIN {X -0.088,Y -244.943,Z 1462.259,A 0.000,B 0.000,C 90.000,E1 46.620} C_DIS
LIN {X -0.086,Y -235.706,Z 1462.238,A 0.000,B 0.000,C 90.000,E1 42.933} C_DIS
LIN {X 0.013,Y -227.400,Z 1462.218,A 0.000,B 0.000,C 90.000,E1 39.152} C_DIS
LIN {X 0.096,Y -220.104,Z 1462.196,A 0.000,B 0.000,C 90.000,E1 35.311} C_DIS
LIN {X -0.022,Y -213.531,Z 1462.175,A 0.000,B 0.000,C 90.000,E1 31.465} C_DIS
LIN {X 0.055,Y -207.825,Z 1462.153,A 0.000,B 0.000,C 90.000,E1 27.513} C_DIS
LIN {X -0.058,Y -202.899,Z 1462.131,A 0.000,B 0.000,C 90.000,E1 23.567} C_DIS
LIN {X 0.029,Y -198.735,Z 1462.109,A 0.000,B 0.000,C 90.000,E1 19.523} C_DIS
LIN {X -0.003,Y -194.718,Z 1462.081,A 0.000,B 0.000,C 90.000,E1 14.662} C_DIS
LIN {X 0.083,Y -191.837,Z 1462.054,A 0.000,B 0.000,C 90.000,E1 9.726} C_DIS
LIN {X -0.032,Y -189.905,Z 1462.027,A 0.000,B 0.000,C 90.000,E1 4.821} C_DIS
LIN {X -0.035,Y -188.812,Z 1461.997,A 0.000,B 0.000,C 90.000,E1 359.542} C_DIS
LIN {X -0.024,Y -188.757,Z 1461.965,A 0.000,B 0.000,C 90.000,E1 353.742} C_DIS
LIN {X 0.016,Y -189.954,Z 1461.933,A 0.000,B 0.000,C 90.000,E1 347.937} C_DIS
LIN {X -0.037,Y -192.622,Z 1461.901,A 0.000,B 0.000,C 90.000,E1 342.181} C_DIS
LIN {X 0.082,Y -196.119,Z 1461.874,A 0.000,B 0.000,C 90.000,E1 337.230} C_DIS
LIN {X 0.035,Y -200.078,Z 1461.851,A 0.000,B 0.000,C 90.000,E1 333.179} C_DIS
LIN {X 0.023,Y -205.195,Z 1461.829,A 0.000,B 0.000,C 90.000,E1 329.154} C_DIS
LIN {X 0.039,Y -210.209,Z 1461.811,A 0.000,B 0.000,C 90.000,E1 325.960} C_DIS
LIN {X -0.099,Y -216.133,Z 1461.793,A 0.000,B 0.000,C 90.000,E1 322.844} C_DIS
LIN {X 0.002,Y -222.956,Z 1461.776,A 0.000,B 0.000,C 90.000,E1 319.703} C_DIS
LIN {X 0.060,Y -230.697,Z 1461.759,A 0.000,B 0.000,C 90.000,E1 316.620} C_DIS
LIN {X -0.026,Y -240.582,Z 1461.740,A 0.000,B 0.000,C 90.000,E1 313.257} C_DIS
LIN {X 0.014,Y -250.513,Z 1461.724,A 0.000,B 0.000,C 90.000,E1 310.297} C_DIS
LIN {X -0.154,Y -261.709,Z 1461.708,A 0.000,B 0.000,C 90.000,E1 307.443} C_DIS
LIN {X -0.134,Y -271.029,Z 1461.696,A 0.000,B 0.000,C 90.000,E1 305.311} C_DIS
LIN {X -0.037,Y -279.695,Z 1461.686,A 0.000,B 0.000,C 90.000,E1 303.547} C_DIS
LIN {X 0.136,Y -289.339,Z 1461.677,A 0.000,B 0.000,C 90.000,E1 301.799} C_DIS
LIN {X 0.069,Y -299.884,Z 1461.667,A 0.000,B 0.000,C 90.000,E1 300.129} C_DIS
LIN {X -0.016,Y -309.214,Z 1461.660,A 0.000,B 0.000,C 90.000,E1 298.821} C_DIS
LIN {X -0.035,Y -317.007,Z 1461.655,A 0.000,B 0.000,C 90.000,E1 297.847} C_DIS
LIN {X -0.050,Y -335.779,Z 1461.643,A 0.000,B 0.000,C 90.000,E1 295.771} C_DIS
LIN {X -0.019,Y -352.394,Z 1461.634,A 0.000,B 0.000,C 90.000,E1 294.079} C_DIS
LIN {X -0.089,Y -363.246,Z 1461.628,A 0.000,B 0.000,C 90.000,E1 293.003} C_DIS
LIN {X 0.065,Y -373.766,Z 1461.622,A 0.000,B 0.000,C 90.000,E1 291.897} C_DIS
LIN {X 0.234,Y -386.809,Z 1461.614,A 0.000,B 0.000,C 90.000,E1 290.482} C_DIS
LIN {X -0.043,Y -394.483,Z 1461.609,A 0.000,B 0.000,C 90.000,E1 289.685} C_DIS
LIN {X -0.136,Y -406.938,Z 1461.602,A 0.000,B 0.000,C 90.000,E1 288.290} C_DIS
LIN {X -0.033,Y -416.328,Z 1461.595,A 0.000,B 0.000,C 90.000,E1 287.166} C_DIS
LIN {X 0.177,Y -422.785,Z 1461.591,A 0.000,B 0.000,C 90.000,E1 286.315} C_DIS
LIN {X -0.079,Y -428.543,Z 1461.586,A 0.000,B 0.000,C 90.000,E1 285.536} C_DIS
LIN {X -0.164,Y -431.898,Z 1461.583,A 0.000,B 0.000,C 90.000,E1 285.009} C_DIS
LIN {X 0.069,Y -436.142,Z 1461.579,A 0.000,B 0.000,C 90.000,E1 284.175} C_DIS
LIN {X -0.185,Y -439.593,Z 1461.574,A 0.000,B 0.000,C 90.000,E1 283.411} C_DIS
LIN {X 0.017,Y -442.350,Z 1461.570,A 0.000,B 0.000,C 90.000,E1 282.591} C_DIS
LIN {X 0.021,Y -443.757,Z 1461.567,A 0.000,B 0.000,C 90.000,E1 282.063} C_DIS
LIN {X 0.033,Y -444.796,Z 1461.564,A 0.000,B 0.000,C 90.000,E1 281.535} C_DIS
LIN {X 0.053,Y -445.339,Z 1461.561,A 0.000,B 0.000,C 90.000,E1 281.007} C_DIS
LIN {X -0.004,Y -445.472,Z 1461.558,A 0.000,B 0.000,C 90.000,E1 280.489} C_DIS
LIN {X 0.025,Y -445.080,Z 1461.555,A 0.000,B 0.000,C 90.000,E1 279.962} C_DIS
LIN {X -0.022,Y -444.180,Z 1461.552,A 0.000,B 0.000,C 90.000,E1 279.443} C_DIS
LIN {X 0.002,Y -442.675,Z 1461.550,A 0.000,B 0.000,C 90.000,E1 278.916} C_DIS
LIN {X -0.049,Y -440.480,Z 1461.547,A 0.000,B 0.000,C 90.000,E1 278.398} C_DIS
LIN {X 0.168,Y -439.134,Z 1461.545,A 0.000,B 0.000,C 90.000,E1 278.106} C_DIS
LIN {X -0.051,Y -437.539,Z 1461.544,A 0.000,B 0.000,C 90.000,E1 277.871} C_DIS
LIN {X -0.129,Y -433.607,Z 1461.541,A 0.000,B 0.000,C 90.000,E1 277.352} C_DIS
LIN {X 0.202,Y -428.476,Z 1461.538,A 0.000,B 0.000,C 90.000,E1 276.777} C_DIS
LIN {X -0.156,Y -422.351,Z 1461.535,A 0.000,B 0.000,C 90.000,E1 276.315} C_DIS
LIN {X 0.018,Y -416.119,Z 1461.532,A 0.000,B 0.000,C 90.000,E1 275.853} C_DIS
LIN {X 0.067,Y -409.413,Z 1461.530,A 0.000,B 0.000,C 90.000,E1 275.454} C_DIS
LIN {X -0.064,Y -399.707,Z 1461.528,A 0.000,B 0.000,C 90.000,E1 274.992} C_DIS
LIN {X 0.193,Y -389.926,Z 1461.525,A 0.000,B 0.000,C 90.000,E1 274.531} C_DIS
LIN {X -0.048,Y -367.923,Z 1461.521,A 0.000,B 0.000,C 90.000,E1 273.726} C_DIS
LIN {X -0.087,Y -358.238,Z 1461.519,A 0.000,B 0.000,C 90.000,E1 273.383} C_DIS
LIN {X 0.098,Y -348.046,Z 1461.517,A 0.000,B 0.000,C 90.000,E1 273.037} C_DIS
LIN {X -0.153,Y -337.506,Z 1461.516,A 0.000,B 0.000,C 90.000,E1 272.808} C_DIS
LIN {X -0.102,Y -326.762,Z 1461.514,A 0.000,B 0.000,C 90.000,E1 272.579} C_DIS
LIN {X 0.129,Y -314.719,Z 1461.513,A 0.000,B 0.000,C 90.000,E1 272.350} C_DIS
LIN {X 0.061,Y -301.325,Z 1461.512,A 0.000,B 0.000,C 90.000,E1 272.236} C_DIS
LIN {X -0.051,Y -293.805,Z 1461.512,A 0.000,B 0.000,C 90.000,E1 272.236} C_DIS
LIN {X -0.066,Y -181.228,Z 1461.512,A 0.000,B 0.000,C 90.000,E1 272.236} C_DIS
LIN {X -0.056,Y -181.565,Z 1461.503,A 0.000,B 0.000,C 90.000,E1 270.516} C_DIS
LIN {X -0.066,Y -181.120,Z 1461.489,A 0.000,B 0.000,C 90.000,E1 267.993} C_DIS
LIN {X -0.077,Y -180.906,Z 1461.475,A 0.000,B 0.000,C 90.000,E1 265.469} C_DIS
LIN {X -0.020,Y -180.725,Z 1461.470,A 0.000,B 0.000,C 90.000,E1 264.609} C_DIS
LIN {X 0.077,Y -178.814,Z 1461.442,A 0.000,B 0.000,C 90.000,E1 259.511} C_DIS
LIN {X -0.016,Y -175.859,Z 1461.414,A 0.000,B 0.000,C 90.000,E1 254.448} C_DIS
LIN {X 0.033,Y -173.824,Z 1461.399,A 0.000,B 0.000,C 90.000,E1 251.873} C_DIS
LIN {X -0.032,Y -171.490,Z 1461.380,A 0.000,B 0.000,C 90.000,E1 248.465} C_DIS
LIN {X -0.045,Y -167.719,Z 1461.356,A 0.000,B 0.000,C 90.000,E1 244.152} C_DIS
LIN {X -0.028,Y -166.411,Z 1461.347,A 0.000,B 0.000,C 90.000,E1 242.410} C_DIS
LIN {X -0.030,Y -163.134,Z 1461.327,A 0.000,B 0.000,C 90.000,E1 238.918} C_DIS
LIN {X -0.064,Y -161.087,Z 1461.313,A 0.000,B 0.000,C 90.000,E1 236.294} C_DIS
LIN {X 0.046,Y -157.817,Z 1461.293,A 0.000,B 0.000,C 90.000,E1 232.718} C_DIS
LIN {X -0.016,Y -155.852,Z 1461.278,A 0.000,B 0.000,C 90.000,E1 230.070} C_DIS
LIN {X 0.040,Y -152.101,Z 1461.253,A 0.000,B 0.000,C 90.000,E1 225.567} C_DIS
LIN {X 0.059,Y -150.352,Z 1461.238,A 0.000,B 0.000,C 90.000,E1 222.852} C_DIS
LIN {X -0.013,Y -147.089,Z 1461.213,A 0.000,B 0.000,C 90.000,E1 218.338} C_DIS
LIN {X -0.018,Y -145.660,Z 1461.198,A 0.000,B 0.000,C 90.000,E1 215.598} C_DIS
LIN {X -0.015,Y -143.042,Z 1461.172,A 0.000,B 0.000,C 90.000,E1 211.003} C_DIS
LIN {X -0.014,Y -141.667,Z 1461.152,A 0.000,B 0.000,C 90.000,E1 207.308} C_DIS
LIN {X 0.030,Y -139.450,Z 1461.116,A 0.000,B 0.000,C 90.000,E1 200.791} C_DIS
LIN {X -0.048,Y -139.184,Z 1461.105,A 0.000,B 0.000,C 90.000,E1 198.960} C_DIS
LIN {X -0.025,Y -138.321,Z 1461.053,A 0.000,B 0.000,C 90.000,E1 189.613} C_DIS
LIN {X -0.018,Y -139.462,Z 1461.007,A 0.000,B 0.000,C 90.000,E1 181.203} C_DIS
LIN {X 0.062,Y -141.020,Z 1460.976,A 0.000,B 0.000,C 90.000,E1 175.584} C_DIS
LIN {X 0.017,Y -142.384,Z 1460.960,A 0.000,B 0.000,C 90.000,E1 172.818} C_DIS
LIN {X -0.062,Y -144.615,Z 1460.934,A 0.000,B 0.000,C 90.000,E1 168.229} C_DIS
LIN {X 0.000,Y -147.809,Z 1460.909,A 0.000,B 0.000,C 90.000,E1 163.614} C_DIS
LIN {X 0.087,Y -150.497,Z 1460.889,A 0.000,B 0.000,C 90.000,E1 159.934} C_DIS
LIN {X -0.034,Y -153.955,Z 1460.869,A 0.000,B 0.000,C 90.000,E1 156.357} C_DIS
LIN {X 0.030,Y -157.366,Z 1460.849,A 0.000,B 0.000,C 90.000,E1 152.743} C_DIS
LIN {X -0.028,Y -161.565,Z 1460.829,A 0.000,B 0.000,C 90.000,E1 149.203} C_DIS
LIN {X -0.016,Y -165.762,Z 1460.809,A 0.000,B 0.000,C 90.000,E1 145.674} C_DIS
LIN {X -0.029,Y -170.719,Z 1460.790,A 0.000,B 0.000,C 90.000,E1 142.190} C_DIS
LIN {X 0.013,Y -175.592,Z 1460.771,A 0.000,B 0.000,C 90.000,E1 138.728} C_DIS
LIN {X 0.000,Y -181.209,Z 1460.752,A 0.000,B 0.000,C 90.000,E1 135.324} C_DIS
LIN {X -0.007,Y -186.674,Z 1460.733,A 0.000,B 0.000,C 90.000,E1 131.962} C_DIS
LIN {X -0.064,Y -191.276,Z 1460.719,A 0.000,B 0.000,C 90.000,E1 129.483} C_DIS
LIN {X 0.016,Y -197.100,Z 1460.701,A 0.000,B 0.000,C 90.000,E1 126.171} C_DIS
LIN {X 0.038,Y -200.865,Z 1460.691,A 0.000,B 0.000,C 90.000,E1 124.278} C_DIS
LIN {X 0.023,Y -312.596,Z 1460.690,A 0.000,B 0.000,C 90.000,E1 124.278} C_DIS
LIN {X -0.058,Y -315.426,Z 1460.690,A 0.000,B 0.000,C 90.000,E1 124.246} C_DIS
LIN {X -0.031,Y -320.176,Z 1460.689,A 0.000,B 0.000,C 90.000,E1 123.992} C_DIS
LIN {X 0.177,Y -322.854,Z 1460.687,A 0.000,B 0.000,C 90.000,E1 123.706} C_DIS
LIN {X -0.021,Y -326.570,Z 1460.684,A 0.000,B 0.000,C 90.000,E1 123.214} C_DIS
LIN {X 0.071,Y -328.126,Z 1460.683,A 0.000,B 0.000,C 90.000,E1 122.880} C_DIS
LIN {X -0.058,Y -341.398,Z 1460.664,A 0.000,B 0.000,C 90.000,E1 119.461} C_DIS
LIN {X 0.016,Y -353.690,Z 1460.648,A 0.000,B 0.000,C 90.000,E1 116.693} C_DIS
LIN {X -0.037,Y -367.465,Z 1460.633,A 0.000,B 0.000,C 90.000,E1 114.003} C_DIS
LIN {X -0.085,Y -381.049,Z 1460.620,A 0.000,B 0.000,C 90.000,E1 111.663} C_DIS
LIN {X 0.089,Y -395.992,Z 1460.608,A 0.000,B 0.000,C 90.000,E1 109.341} C_DIS
LIN {X 0.128,Y -412.396,Z 1460.595,A 0.000,B 0.000,C 90.000,E1 107.094} C_DIS
LIN {X -0.207,Y -430.379,Z 1460.583,A 0.000,B 0.000,C 90.000,E1 104.954} C_DIS
LIN {X -0.100,Y -449.906,Z 1460.571,A 0.000,B 0.000,C 90.000,E1 102.827} C_DIS
LIN {X 0.199,Y -470.150,Z 1460.560,A 0.000,B 0.000,C 90.000,E1 100.838} C_DIS
LIN {X 0.173,Y -488.202,Z 1460.552,A 0.000,B 0.000,C 90.000,E1 99.265} C_DIS
LIN {X -0.157,Y -490.183,Z 1460.550,A 0.000,B 0.000,C 90.000,E1 99.086} C_DIS
LIN {X 0.152,Y -491.882,Z 1460.549,A 0.000,B 0.000,C 90.000,E1 98.803} C_DIS
LIN {X 0.051,Y -493.153,Z 1460.548,A 0.000,B 0.000,C 90.000,E1 98.568} C_DIS
LIN {X -0.205,Y -494.709,Z 1460.545,A 0.000,B 0.000,C 90.000,E1 98.106} C_DIS
LIN {X 0.037,Y -495.191,Z 1460.542,A 0.000,B 0.000,C 90.000,E1 97.587} C_DIS
LIN {X -0.200,Y -494.683,Z 1460.539,A 0.000,B 0.000,C 90.000,E1 97.125} C_DIS
LIN {X 0.055,Y -493.104,Z 1460.537,A 0.000,B 0.000,C 90.000,E1 96.606} C_DIS
LIN {X -0.036,Y -491.827,Z 1460.535,A 0.000,B 0.000,C 90.000,E1 96.372} C_DIS
LIN {X -0.200,Y -478.611,Z 1460.524,A 0.000,B 0.000,C 90.000,E1 94.416} C_DIS
LIN {X 0.186,Y -469.514,Z 1460.516,A 0.000,B 0.000,C 90.000,E1 92.865} C_DIS
LIN {X -0.140,Y -463.082,Z 1460.510,A 0.000,B 0.000,C 90.000,E1 91.892} C_DIS
LIN {X 0.173,Y -451.244,Z 1460.500,A 0.000,B 0.000,C 90.000,E1 90.057} C_DIS
LIN {X -0.128,Y -434.434,Z 1460.486,A 0.000,B 0.000,C 90.000,E1 87.478} C_DIS
LIN {X 0.047,Y -422.653,Z 1460.475,A 0.000,B 0.000,C 90.000,E1 85.584} C_DIS
LIN {X -0.066,Y -412.618,Z 1460.466,A 0.000,B 0.000,C 90.000,E1 83.970} C_DIS
LIN {X 0.149,Y -400.713,Z 1460.456,A 0.000,B 0.000,C 90.000,E1 82.008} C_DIS
LIN {X -0.172,Y -386.979,Z 1460.443,A 0.000,B 0.000,C 90.000,E1 79.803} C_DIS
LIN {X 0.084,Y -371.881,Z 1460.429,A 0.000,B 0.000,C 90.000,E1 77.173} C_DIS
LIN {X 0.074,Y -360.595,Z 1460.417,A 0.000,B 0.000,C 90.000,E1 75.117} C_DIS
LIN {X 0.070,Y -350.891,Z 1460.407,A 0.000,B 0.000,C 90.000,E1 73.323} C_DIS
LIN {X -0.101,Y -339.488,Z 1460.396,A 0.000,B 0.000,C 90.000,E1 71.221} C_DIS
LIN {X 0.029,Y -328.301,Z 1460.384,A 0.000,B 0.000,C 90.000,E1 69.028} C_DIS
LIN {X 0.002,Y -311.545,Z 1460.364,A 0.000,B 0.000,C 90.000,E1 65.537} C_DIS
LIN {X -0.051,Y -297.405,Z 1460.346,A 0.000,B 0.000,C 90.000,E1 62.281} C_DIS
LIN {X 0.023,Y -284.389,Z 1460.327,A 0.000,B 0.000,C 90.000,E1 58.918} C_DIS
LIN {X -0.133,Y -274.582,Z 1460.312,A 0.000,B 0.000,C 90.000,E1 56.215} C_DIS
LIN {X 0.056,Y -262.855,Z 1460.293,A 0.000,B 0.000,C 90.000,E1 52.683} C_DIS
LIN {X 0.120,Y -253.062,Z 1460.275,A 0.000,B 0.000,C 90.000,E1 49.461} C_DIS
LIN {X -0.140,Y -243.113,Z 1460.255,A 0.000,B 0.000,C 90.000,E1 45.891} C_DIS
LIN {X -0.018,Y -234.079,Z 1460.234,A 0.000,B 0.000,C 90.000,E1 42.162} C_DIS
LIN {X 0.026,Y -226.040,Z 1460.213,A 0.000,B 0.000,C 90.000,E1 38.382} C_DIS
LIN {X 0.102,Y -218.894,Z 1460.192,A 0.000,B 0.000,C 90.000,E1 34.532} C_DIS
LIN {X 0.011,Y -212.489,Z 1460.170,A 0.000,B 0.000,C 90.000,E1 30.669} C_DIS
LIN {X -0.042,Y -206.952,Z 1460.149,A 0.000,B 0.000,C 90.000,E1 26.744} C_DIS
LIN {X -0.078,Y -202.191,Z 1460.126,A 0.000,B 0.000,C 90.000,E1 22.770} C_DIS
LIN {X -0.052,Y -197.489,Z 1460.099,A 0.000,B 0.000,C 90.000,E1 17.928} C_DIS
LIN {X 0.078,Y -193.897,Z 1460.072,A 0.000,B 0.000,C 90.000,E1 13.008} C_DIS
LIN {X -0.020,Y -191.041,Z 1460.041,A 0.000,B 0.000,C 90.000,E1 7.296} C_DIS
LIN {X 0.089,Y -189.390,Z 1460.008,A 0.000,B 0.000,C 90.000,E1 1.489} C_DIS
LIN {X -0.061,Y -188.910,Z 1459.974,A 0.000,B 0.000,C 90.000,E1 355.412} C_DIS
LIN {X -0.107,Y -189.702,Z 1459.942,A 0.000,B 0.000,C 90.000,E1 349.634} C_DIS
LIN {X -0.045,Y -192.326,Z 1459.906,A 0.000,B 0.000,C 90.000,E1 343.015} C_DIS
LIN {X -0.070,Y -195.612,Z 1459.878,A 0.000,B 0.000,C 90.000,E1 338.103} C_DIS
LIN {X -0.045,Y -199.342,Z 1459.856,A 0.000,B 0.000,C 90.000,E1 334.024} C_DIS
LIN {X -0.081,Y -204.235,Z 1459.833,A 0.000,B 0.000,C 90.000,E1 329.999} C_DIS
LIN {X -0.022,Y -209.028,Z 1459.815,A 0.000,B 0.000,C 90.000,E1 326.786} C_DIS
LIN {X -0.018,Y -214.714,Z 1459.798,A 0.000,B 0.000,C 90.000,E1 323.623} C_DIS
LIN {X -0.086,Y -221.305,Z 1459.781,A 0.000,B 0.000,C 90.000,E1 320.517} C_DIS
LIN {X 0.097,Y -228.807,Z 1459.763,A 0.000,B 0.000,C 90.000,E1 317.391} C_DIS
LIN {X -0.049,Y -238.448,Z 1459.745,A 0.000,B 0.000,C 90.000,E1 314.028} C_DIS
LIN {X -0.066,Y -248.065,Z 1459.728,A 0.000,B 0.000,C 90.000,E1 311.067} C_DIS
LIN {X -0.135,Y -258.936,Z 1459.712,A 0.000,B 0.000,C 90.000,E1 308.177} C_DIS
LIN {X 0.052,Y -269.542,Z 1459.698,A 0.000,B 0.000,C 90.000,E1 305.644} C_DIS
LIN {X -0.085,Y -279.792,Z 1459.686,A 0.000,B 0.000,C 90.000,E1 303.579} C_DIS
LIN {X -0.150,Y -289.395,Z 1459.677,A 0.000,B 0.000,C 90.000,E1 301.878} C_DIS
LIN {X 0.186,Y -299.932,Z 1459.668,A 0.000,B 0.000,C 90.000,E1 300.129} C_DIS
LIN {X 0.106,Y -309.255,Z 1459.660,A 0.000,B 0.000,C 90.000,E1 298.821} C_DIS
LIN {X 0.140,Y -316.968,Z 1459.655,A 0.000,B 0.000,C 90.000,E1 297.847} C_DIS
LIN {X 0.020,Y -335.619,Z 1459.643,A 0.000,B 0.000,C 90.000,E1 295.796} C_DIS
LIN {X 0.000,Y -352.041,Z 1459.634,A 0.000,B 0.000,C 90.000,E1 294.131} C_DIS
LIN {X 0.085,Y -362.939,Z 1459.628,A 0.000,B 0.000,C 90.000,E1 293.025} C_DIS
LIN {X 0.147,Y -370.908,Z 1459.624,A 0.000,B 0.000,C 90.000,E1 292.206} C_DIS
LIN {X -0.028,Y -383.948,Z 1459.616,A 0.000,B 0.000,C 90.000,E1 290.844} C_DIS
LIN {X -0.213,Y -394.174,Z 1459.610,A 0.000,B 0.000,C 90.000,E1 289.758} C_DIS
LIN {X 0.072,Y -406.653,Z 1459.602,A 0.000,B 0.000,C 90.000,E1 288.308} C_DIS
LIN {X -0.089,Y -416.106,Z 1459.596,A 0.000,B 0.000,C 90.000,E1 287.221} C_DIS
LIN {X -0.003,Y -422.646,Z 1459.591,A 0.000,B 0.000,C 90.000,E1 286.386} C_DIS
LIN {X 0.154,Y -428.477,Z 1459.587,A 0.000,B 0.000,C 90.000,E1 285.552} C_DIS
LIN {X 0.187,Y -431.872,Z 1459.583,A 0.000,B 0.000,C 90.000,E1 285.009} C_DIS
LIN {X -0.107,Y -436.191,Z 1459.579,A 0.000,B 0.000,C 90.000,E1 284.245} C_DIS
LIN {X 0.171,Y -439.689,Z 1459.575,A 0.000,B 0.000,C 90.000,E1 283.411} C_DIS
LIN {X -0.054,Y -442.492,Z 1459.570,A 0.000,B 0.000,C 90.000,E1 282.647} C_DIS
LIN {X -0.052,Y -443.918,Z 1459.567,A 0.000,B 0.000,C 90.000,E1 282.119} C_DIS
LIN {X -0.038,Y -445.002,Z 1459.564,A 0.000,B 0.000,C 90.000,E1 281.591} C_DIS
LIN {X -0.104,Y -445.637,Z 1459.561,A 0.000,B 0.000,C 90.000,E1 281.074} C_DIS
LIN {X -0.076,Y -445.805,Z 1459.559,A 0.000,B 0.000,C 90.000,E1 280.546} C_DIS
LIN {X -0.046,Y -445.463,Z 1459.556,A 0.000,B 0.000,C 90.000,E1 280.018} C_DIS
LIN {X -0.092,Y -444.637,Z 1459.553,A 0.000,B 0.000,C 90.000,E1 279.500} C_DIS
LIN {X -0.066,Y -443.229,Z 1459.550,A 0.000,B 0.000,C 90.000,E1 278.973} C_DIS
LIN {X -0.115,Y -441.174,Z 1459.547,A 0.000,B 0.000,C 90.000,E1 278.454} C_DIS
LIN {X -0.168,Y -438.331,Z 1459.544,A 0.000,B 0.000,C 90.000,E1 277.936} C_DIS
LIN {X -0.182,Y -434.528,Z 1459.541,A 0.000,B 0.000,C 90.000,E1 277.409} C_DIS
LIN {X 0.155,Y -429.616,Z 1459.538,A 0.000,B 0.000,C 90.000,E1 276.834} C_DIS
LIN {X 0.149,Y -423.536,Z 1459.535,A 0.000,B 0.000,C 90.000,E1 276.315} C_DIS
LIN {X -0.139,Y -417.355,Z 1459.533,A 0.000,B 0.000,C 90.000,E1 275.910} C_DIS
LIN {X -0.123,Y -410.688,Z 1459.531,A 0.000,B 0.000,C 90.000,E1 275.511} C_DIS
LIN {X 0.091,Y -400.984,Z 1459.528,A 0.000,B 0.000,C 90.000,E1 274.992} C_DIS
LIN {X -0.074,Y -391.192,Z 1459.525,A 0.000,B 0.000,C 90.000,E1 274.588} C_DIS
LIN {X 0.066,Y -372.197,Z 1459.521,A 0.000,B 0.000,C 90.000,E1 273.841} C_DIS
LIN {X -0.015,Y -359.385,Z 1459.519,A 0.000,B 0.000,C 90.000,E1 273.383} C_DIS
LIN {X 0.153,Y -349.234,Z 1459.517,A 0.000,B 0.000,C 90.000,E1 273.037} C_DIS
LIN {X 0.118,Y -335.416,Z 1459.515,A 0.000,B 0.000,C 90.000,E1 272.694} C_DIS
LIN {X -0.140,Y -323.961,Z 1459.514,A 0.000,B 0.000,C 90.000,E1 272.522} C_DIS
LIN {X 0.154,Y -315.925,Z 1459.513,A 0.000,B 0.000,C 90.000,E1 272.350} C_DIS
LIN {X 0.083,Y -302.398,Z 1459.512,A 0.000,B 0.000,C 90.000,E1 272.236} C_DIS
LIN {X -0.029,Y -297.315,Z 1459.512,A 0.000,B 0.000,C 90.000,E1 272.236} C_DIS
LIN {X -0.052,Y -181.227,Z 1459.512,A 0.000,B 0.000,C 90.000,E1 272.236} C_DIS
LIN {X -0.041,Y -181.565,Z 1459.503,A 0.000,B 0.000,C 90.000,E1 270.516} C_DIS
LIN {X -0.051,Y -181.121,Z 1459.489,A 0.000,B 0.000,C 90.000,E1 267.993} C_DIS
LIN {X -0.062,Y -180.906,Z 1459.475,A 0.000,B 0.000,C 90.000,E1 265.469} C_DIS
LIN {X -0.006,Y -180.727,Z 1459.470,A 0.000,B 0.000,C 90.000,E1 264.609} C_DIS
LIN {X 0.092,Y -178.817,Z 1459.442,A 0.000,B 0.000,C 90.000,E1 259.511} C_DIS
LIN {X -0.001,Y -175.861,Z 1459.414,A 0.000,B 0.000,C 90.000,E1 254.448} C_DIS
LIN {X 0.047,Y -173.827,Z 1459.399,A 0.000,B 0.000,C 90.000,E1 251.873} C_DIS
LIN {X -0.018,Y -171.494,Z 1459.380,A 0.000,B 0.000,C 90.000,E1 248.465} C_DIS
LIN {X -0.030,Y -167.723,Z 1459.356,A 0.000,B 0.000,C 90.000,E1 244.152} C_DIS
LIN {X -0.014,Y -166.416,Z 1459.347,A 0.000,B 0.000,C 90.000,E1 242.410} C_DIS
LIN {X -0.015,Y -163.138,Z 1459.327,A 0.000,B 0.000,C 90.000,E1 238.918} C_DIS
LIN {X -0.050,Y -161.092,Z 1459.313,A 0.000,B 0.000,C 90.000,E1 236.294} C_DIS
LIN {X -0.066,Y -157.821,Z 1459.293,A 0.000,B 0.000,C 90.000,E1 232.763} C_DIS
LIN {X -0.002,Y -155.855,Z 1459.278,A 0.000,B 0.000,C 90.000,E1 230.070} C_DIS
LIN {X 0.053,Y -152.105,Z 1459.253,A 0.000,B 0.000,C 90.000,E1 225.567} C_DIS
LIN {X 0.072,Y -150.355,Z 1459.238,A 0.000,B 0.000,C 90.000,E1 222.852} C_DIS
LIN {X 0.000,Y -147.091,Z 1459.213,A 0.000,B 0.000,C 90.000,E1 218.338} C_DIS
LIN {X -0.006,Y -145.662,Z 1459.198,A 0.000,B 0.000,C 90.000,E1 215.598} C_DIS
LIN {X -0.002,Y -143.044,Z 1459.172,A 0.000,B 0.000,C 90.000,E1 211.003} C_DIS
LIN {X -0.001,Y -141.669,Z 1459.152,A 0.000,B 0.000,C 90.000,E1 207.308} C_DIS
LIN {X 0.043,Y -139.451,Z 1459.116,A 0.000,B 0.000,C 90.000,E1 200.791} C_DIS
LIN {X -0.036,Y -139.185,Z 1459.105,A 0.000,B 0.000,C 90.000,E1 198.960} C_DIS
LIN {X -0.013,Y -138.322,Z 1459.053,A 0.000,B 0.000,C 90.000,E1 189.613} C_DIS
LIN {X -0.006,Y -139.461,Z 1459.007,A 0.000,B 0.000,C 90.000,E1 181.203} C_DIS
LIN {X -0.066,Y -141.018,Z 1458.976,A 0.000,B 0.000,C 90.000,E1 175.641} C_DIS
LIN {X 0.030,Y -142.381,Z 1458.960,A 0.000,B 0.000,C 90.000,E1 172.818} C_DIS
LIN {X -0.049,Y -144.612,Z 1458.934,A 0.000,B 0.000,C 90.000,E1 168.229} C_DIS
LIN {X 0.012,Y -147.806,Z 1458.909,A 0.000,B 0.000,C 90.000,E1 163.614} C_DIS
LIN {X -0.093,Y -150.492,Z 1458.889,A 0.000,B 0.000,C 90.000,E1 160.007} C_DIS
LIN {X -0.019,Y -153.949,Z 1458.869,A 0.000,B 0.000,C 90.000,E1 156.357} C_DIS
LIN {X 0.043,Y -157.360,Z 1458.849,A 0.000,B 0.000,C 90.000,E1 152.743} C_DIS
LIN {X -0.014,Y -161.559,Z 1458.829,A 0.000,B 0.000,C 90.000,E1 149.203} C_DIS
LIN {X -0.002,Y -165.756,Z 1458.809,A 0.000,B 0.000,C 90.000,E1 145.674} C_DIS
LIN {X -0.015,Y -170.712,Z 1458.790,A 0.000,B 0.000,C 90.000,E1 142.190} C_DIS
LIN {X 0.028,Y -175.584,Z 1458.771,A 0.000,B 0.000,C 90.000,E1 138.728} C_DIS
LIN {X 0.015,Y -181.203,Z 1458.752,A 0.000,B 0.000,C 90.000,E1 135.324} C_DIS
LIN {X 0.007,Y -186.665,Z 1458.733,A 0.000,B 0.000,C 90.000,E1 131.962} C_DIS
LIN {X -0.049,Y -191.269,Z 1458.719,A 0.000,B 0.000,C 90.000,E1 129.483} C_DIS
LIN {X 0.031,Y -197.091,Z 1458.701,A 0.000,B 0.000,C 90.000,E1 126.171} C_DIS
LIN {X -0.028,Y -200.814,Z 1458.691,A 0.000,B 0.000,C 90.000,E1 124.326} C_DIS
LIN {X -0.091,Y -312.675,Z 1458.691,A 0.000,B 0.000,C 90.000,E1 124.326} C_DIS
LIN {X -0.211,Y -317.788,Z 1458.690,A 0.000,B 0.000,C 90.000,E1 124.199} C_DIS
LIN {X 0.162,Y -319.961,Z 1458.689,A 0.000,B 0.000,C 90.000,E1 123.992} C_DIS
LIN {X 0.202,Y -322.938,Z 1458.688,A 0.000,B 0.000,C 90.000,E1 123.706} C_DIS
LIN {X -0.014,Y -326.594,Z 1458.684,A 0.000,B 0.000,C 90.000,E1 123.214} C_DIS
LIN {X 0.077,Y -328.120,Z 1458.683,A 0.000,B 0.000,C 90.000,E1 122.880} C_DIS
LIN {X -0.052,Y -341.372,Z 1458.664,A 0.000,B 0.000,C 90.000,E1 119.461} C_DIS
LIN {X 0.022,Y -353.663,Z 1458.648,A 0.000,B 0.000,C 90.000,E1 116.693} C_DIS
LIN {X -0.033,Y -367.438,Z 1458.633,A 0.000,B 0.000,C 90.000,E1 114.003} C_DIS
LIN {X -0.080,Y -381.020,Z 1458.620,A 0.000,B 0.000,C 90.000,E1 111.663} C_DIS
LIN {X 0.093,Y -395.962,Z 1458.608,A 0.000,B 0.000,C 90.000,E1 109.341} C_DIS
LIN {X 0.132,Y -412.366,Z 1458.595,A 0.000,B 0.000,C 90.000,E1 107.094} C_DIS
LIN {X -0.204,Y -430.348,Z 1458.583,A 0.000,B 0.000,C 90.000,E1 104.954} C_DIS
LIN {X -0.098,Y -449.875,Z 1458.571,A 0.000,B 0.000,C 90.000,E1 102.827} C_DIS
LIN {X 0.200,Y -470.118,Z 1458.560,A 0.000,B 0.000,C 90.000,E1 100.838} C_DIS
LIN {X 0.173,Y -488.161,Z 1458.552,A 0.000,B 0.000,C 90.000,E1 99.265} C_DIS
LIN {X -0.157,Y -490.124,Z 1458.550,A 0.000,B 0.000,C 90.000,E1 99.086} C_DIS
LIN {X 0.152,Y -491.808,Z 1458.549,A 0.000,B 0.000,C 90.000,E1 98.803} C_DIS
LIN {X 0.051,Y -493.068,Z 1458.548,A 0.000,B 0.000,C 90.000,E1 98.568} C_DIS
LIN {X -0.205,Y -494.607,Z 1458.545,A 0.000,B 0.000,C 90.000,E1 98.106} C_DIS
LIN {X 0.036,Y -495.075,Z 1458.542,A 0.000,B 0.000,C 90.000,E1 97.587} C_DIS
LIN {X -0.202,Y -494.553,Z 1458.539,A 0.000,B 0.000,C 90.000,E1 97.125} C_DIS
LIN {X 0.053,Y -492.958,Z 1458.537,A 0.000,B 0.000,C 90.000,E1 96.606} C_DIS
LIN {X -0.039,Y -491.670,Z 1458.535,A 0.000,B 0.000,C 90.000,E1 96.372} C_DIS
LIN {X -0.207,Y -478.452,Z 1458.524,A 0.000,B 0.000,C 90.000,E1 94.416} C_DIS
LIN {X 0.178,Y -469.351,Z 1458.516,A 0.000,B 0.000,C 90.000,E1 92.865} C_DIS
LIN {X -0.151,Y -462.901,Z 1458.510,A 0.000,B 0.000,C 90.000,E1 91.892} C_DIS
LIN {X -0.064,Y -452.755,Z 1458.502,A 0.000,B 0.000,C 90.000,E1 90.344} C_DIS
LIN {X 0.122,Y -435.945,Z 1458.487,A 0.000,B 0.000,C 90.000,E1 87.707} C_DIS
LIN {X 0.172,Y -425.898,Z 1458.479,A 0.000,B 0.000,C 90.000,E1 86.102} C_DIS
LIN {X 0.198,Y -414.209,Z 1458.468,A 0.000,B 0.000,C 90.000,E1 84.204} C_DIS
LIN {X -0.067,Y -404.087,Z 1458.459,A 0.000,B 0.000,C 90.000,E1 82.591} C_DIS
LIN {X 0.008,Y -392.082,Z 1458.448,A 0.000,B 0.000,C 90.000,E1 80.622} C_DIS
LIN {X 0.002,Y -378.544,Z 1458.435,A 0.000,B 0.000,C 90.000,E1 78.342} C_DIS
LIN {X 0.082,Y -362.237,Z 1458.419,A 0.000,B 0.000,C 90.000,E1 75.408} C_DIS
LIN {X 0.051,Y -350.925,Z 1458.407,A 0.000,B 0.000,C 90.000,E1 73.323} C_DIS
LIN {X -0.119,Y -339.517,Z 1458.396,A 0.000,B 0.000,C 90.000,E1 71.221} C_DIS
LIN {X -0.018,Y -326.695,Z 1458.382,A 0.000,B 0.000,C 90.000,E1 68.720} C_DIS
LIN {X -0.014,Y -311.507,Z 1458.364,A 0.000,B 0.000,C 90.000,E1 65.537} C_DIS
LIN {X -0.068,Y -297.360,Z 1458.346,A 0.000,B 0.000,C 90.000,E1 62.281} C_DIS
LIN {X 0.005,Y -284.346,Z 1458.327,A 0.000,B 0.000,C 90.000,E1 58.918} C_DIS
LIN {X 0.174,Y -273.369,Z 1458.310,A 0.000,B 0.000,C 90.000,E1 55.801} C_DIS
LIN {X -0.058,Y -261.725,Z 1458.291,A 0.000,B 0.000,C 90.000,E1 52.351} C_DIS
LIN {X -0.022,Y -251.053,Z 1458.271,A 0.000,B 0.000,C 90.000,E1 48.771} C_DIS
LIN {X 0.003,Y -241.357,Z 1458.251,A 0.000,B 0.000,C 90.000,E1 45.121} C_DIS
LIN {X 0.070,Y -232.534,Z 1458.230,A 0.000,B 0.000,C 90.000,E1 41.391} C_DIS
LIN {X -0.081,Y -224.716,Z 1458.209,A 0.000,B 0.000,C 90.000,E1 37.649} C_DIS
LIN {X 0.008,Y -217.725,Z 1458.188,A 0.000,B 0.000,C 90.000,E1 33.785} C_DIS
LIN {X 0.068,Y -211.490,Z 1458.166,A 0.000,B 0.000,C 90.000,E1 29.873} C_DIS
LIN {X 0.071,Y -206.123,Z 1458.144,A 0.000,B 0.000,C 90.000,E1 25.924} C_DIS
LIN {X -0.070,Y -201.546,Z 1458.122,A 0.000,B 0.000,C 90.000,E1 21.972} C_DIS
LIN {X 0.056,Y -197.035,Z 1458.095,A 0.000,B 0.000,C 90.000,E1 17.094} C_DIS
LIN {X -0.064,Y -193.665,Z 1458.068,A 0.000,B 0.000,C 90.000,E1 12.243} C_DIS
LIN {X -0.016,Y -191.018,Z 1458.036,A 0.000,B 0.000,C 90.000,E1 6.486} C_DIS
LIN {X 0.000,Y -189.411,Z 1458.000,A 0.000,B 0.000,C 90.000,E1 360.000} C_DIS
LIN {X 0.057,Y -189.204,Z 1457.970,A 0.000,B 0.000,C 90.000,E1 354.552} C_DIS
LIN {X 0.079,Y -190.158,Z 1457.938,A 0.000,B 0.000,C 90.000,E1 348.757} C_DIS
LIN {X 0.026,Y -192.972,Z 1457.901,A 0.000,B 0.000,C 90.000,E1 342.181} C_DIS
LIN {X -0.022,Y -196.437,Z 1457.874,A 0.000,B 0.000,C 90.000,E1 337.283} C_DIS
LIN {X 0.034,Y -200.379,Z 1457.851,A 0.000,B 0.000,C 90.000,E1 333.204} C_DIS
LIN {X -0.052,Y -205.501,Z 1457.829,A 0.000,B 0.000,C 90.000,E1 329.203} C_DIS
LIN {X -0.024,Y -210.502,Z 1457.811,A 0.000,B 0.000,C 90.000,E1 326.008} C_DIS
LIN {X 0.022,Y -216.414,Z 1457.794,A 0.000,B 0.000,C 90.000,E1 322.844} C_DIS
LIN {X -0.036,Y -223.238,Z 1457.776,A 0.000,B 0.000,C 90.000,E1 319.747} C_DIS
LIN {X 0.036,Y -231.005,Z 1457.759,A 0.000,B 0.000,C 90.000,E1 316.662} C_DIS
LIN {X -0.042,Y -240.875,Z 1457.740,A 0.000,B 0.000,C 90.000,E1 313.299} C_DIS
LIN {X 0.027,Y -250.824,Z 1457.724,A 0.000,B 0.000,C 90.000,E1 310.334} C_DIS
LIN {X 0.037,Y -262.006,Z 1457.708,A 0.000,B 0.000,C 90.000,E1 307.443} C_DIS
LIN {X -0.015,Y -272.947,Z 1457.694,A 0.000,B 0.000,C 90.000,E1 304.978} C_DIS
LIN {X -0.030,Y -281.716,Z 1457.685,A 0.000,B 0.000,C 90.000,E1 303.245} C_DIS
LIN {X -0.067,Y -291.484,Z 1457.675,A 0.000,B 0.000,C 90.000,E1 301.544} C_DIS
LIN {X -0.099,Y -302.212,Z 1457.666,A 0.000,B 0.000,C 90.000,E1 299.873} C_DIS
LIN {X -0.044,Y -309.296,Z 1457.660,A 0.000,B 0.000,C 90.000,E1 298.871} C_DIS
LIN {X -0.047,Y -319.648,Z 1457.653,A 0.000,B 0.000,C 90.000,E1 297.590} C_DIS
LIN {X 0.007,Y -336.071,Z 1457.643,A 0.000,B 0.000,C 90.000,E1 295.771} C_DIS
LIN {X -0.100,Y -349.892,Z 1457.635,A 0.000,B 0.000,C 90.000,E1 294.387} C_DIS
LIN {X -0.028,Y -363.532,Z 1457.628,A 0.000,B 0.000,C 90.000,E1 293.003} C_DIS
LIN {X 0.062,Y -374.097,Z 1457.622,A 0.000,B 0.000,C 90.000,E1 291.897} C_DIS
LIN {X -0.078,Y -386.842,Z 1457.614,A 0.000,B 0.000,C 90.000,E1 290.556} C_DIS
LIN {X -0.037,Y -396.851,Z 1457.608,A 0.000,B 0.000,C 90.000,E1 289.450} C_DIS
LIN {X -0.114,Y -409.246,Z 1457.600,A 0.000,B 0.000,C 90.000,E1 288.055} C_DIS
LIN {X 0.145,Y -418.567,Z 1457.594,A 0.000,B 0.000,C 90.000,E1 286.913} C_DIS
LIN {X -0.146,Y -424.888,Z 1457.589,A 0.000,B 0.000,C 90.000,E1 286.134} C_DIS
LIN {X 0.158,Y -428.701,Z 1457.587,A 0.000,B 0.000,C 90.000,E1 285.552} C_DIS
LIN {X 0.192,Y -432.118,Z 1457.583,A 0.000,B 0.000,C 90.000,E1 285.009} C_DIS
LIN {X -0.100,Y -436.447,Z 1457.579,A 0.000,B 0.000,C 90.000,E1 284.245} C_DIS
LIN {X 0.180,Y -439.946,Z 1457.575,A 0.000,B 0.000,C 90.000,E1 283.411} C_DIS
LIN {X -0.043,Y -442.750,Z 1457.570,A 0.000,B 0.000,C 90.000,E1 282.647} C_DIS
LIN {X -0.039,Y -444.205,Z 1457.567,A 0.000,B 0.000,C 90.000,E1 282.119} C_DIS
LIN {X -0.024,Y -445.266,Z 1457.564,A 0.000,B 0.000,C 90.000,E1 281.591} C_DIS
LIN {X -0.089,Y -445.946,Z 1457.561,A 0.000,B 0.000,C 90.000,E1 281.074} C_DIS
LIN {X -0.058,Y -446.117,Z 1457.559,A 0.000,B 0.000,C 90.000,E1 280.546} C_DIS
LIN {X -0.026,Y -445.846,Z 1457.556,A 0.000,B 0.000,C 90.000,E1 280.018} C_DIS
LIN {X -0.071,Y -445.029,Z 1457.553,A 0.000,B 0.000,C 90.000,E1 279.500} C_DIS
LIN {X -0.043,Y -443.642,Z 1457.550,A 0.000,B 0.000,C 90.000,E1 278.973} C_DIS
LIN {X -0.090,Y -441.621,Z 1457.547,A 0.000,B 0.000,C 90.000,E1 278.454} C_DIS
LIN {X -0.141,Y -438.817,Z 1457.544,A 0.000,B 0.000,C 90.000,E1 277.936} C_DIS
LIN {X -0.152,Y -435.111,Z 1457.541,A 0.000,B 0.000,C 90.000,E1 277.409} C_DIS
LIN {X 0.188,Y -430.270,Z 1457.538,A 0.000,B 0.000,C 90.000,E1 276.834} C_DIS
LIN {X 0.123,Y -424.183,Z 1457.535,A 0.000,B 0.000,C 90.000,E1 276.315} C_DIS
LIN {X 0.214,Y -417.826,Z 1457.533,A 0.000,B 0.000,C 90.000,E1 275.853} C_DIS
LIN {X -0.117,Y -411.398,Z 1457.531,A 0.000,B 0.000,C 90.000,E1 275.511} C_DIS
LIN {X -0.069,Y -404.861,Z 1457.529,A 0.000,B 0.000,C 90.000,E1 275.163} C_DIS
LIN {X 0.098,Y -395.333,Z 1457.526,A 0.000,B 0.000,C 90.000,E1 274.702} C_DIS
LIN {X 0.103,Y -385.406,Z 1457.524,A 0.000,B 0.000,C 90.000,E1 274.302} C_DIS
LIN {X -0.009,Y -363.431,Z 1457.519,A 0.000,B 0.000,C 90.000,E1 273.498} C_DIS
LIN {X 0.053,Y -353.401,Z 1457.518,A 0.000,B 0.000,C 90.000,E1 273.154} C_DIS
LIN {X 0.087,Y -343.136,Z 1457.516,A 0.000,B 0.000,C 90.000,E1 272.865} C_DIS
LIN {X 0.000,Y -332.498,Z 1457.515,A 0.000,B 0.000,C 90.000,E1 272.636} C_DIS
LIN {X -0.143,Y -321.019,Z 1457.514,A 0.000,B 0.000,C 90.000,E1 272.465} C_DIS
LIN {X -0.125,Y -312.002,Z 1457.513,A 0.000,B 0.000,C 90.000,E1 272.350} C_DIS
LIN {X 0.093,Y -303.215,Z 1457.513,A 0.000,B 0.000,C 90.000,E1 272.236} C_DIS
LIN {X -0.020,Y -298.239,Z 1457.512,A 0.000,B 0.000,C 90.000,E1 272.236} C_DIS
LIN {X -0.047,Y -181.227,Z 1457.512,A 0.000,B 0.000,C 90.000,E1 272.236} C_DIS
LIN {X -0.036,Y -181.564,Z 1457.503,A 0.000,B 0.000,C 90.000,E1 270.516} C_DIS
LIN {X -0.046,Y -181.121,Z 1457.489,A 0.000,B 0.000,C 90.000,E1 267.993} C_DIS
LIN {X -0.057,Y -180.907,Z 1457.475,A 0.000,B 0.000,C 90.000,E1 265.469} C_DIS
LIN {X -0.001,Y -180.729,Z 1457.470,A 0.000,B 0.000,C 90.000,E1 264.609} C_DIS
LIN {X 0.097,Y -178.817,Z 1457.442,A 0.000,B 0.000,C 90.000,E1 259.511} C_DIS
LIN {X 0.003,Y -175.862,Z 1457.414,A 0.000,B 0.000,C 90.000,E1 254.448} C_DIS
LIN {X 0.052,Y -173.828,Z 1457.399,A 0.000,B 0.000,C 90.000,E1 251.873} C_DIS
LIN {X -0.013,Y -171.496,Z 1457.380,A 0.000,B 0.000,C 90.000,E1 248.465} C_DIS
LIN {X -0.026,Y -167.724,Z 1457.356,A 0.000,B 0.000,C 90.000,E1 244.152} C_DIS
LIN {X -0.009,Y -166.418,Z 1457.347,A 0.000,B 0.000,C 90.000,E1 242.410} C_DIS
LIN {X -0.011,Y -163.139,Z 1457.327,A 0.000,B 0.000,C 90.000,E1 238.918} C_DIS
LIN {X -0.046,Y -161.094,Z 1457.313,A 0.000,B 0.000,C 90.000,E1 236.294} C_DIS
LIN {X -0.062,Y -157.823,Z 1457.293,A 0.000,B 0.000,C 90.000,E1 232.763} C_DIS
LIN {X 0.002,Y -155.857,Z 1457.278,A 0.000,B 0.000,C 90.000,E1 230.070} C_DIS
LIN {X 0.057,Y -152.106,Z 1457.253,A 0.000,B 0.000,C 90.000,E1 225.567} C_DIS
LIN {X 0.076,Y -150.357,Z 1457.238,A 0.000,B 0.000,C 90.000,E1 222.852} C_DIS
LIN {X 0.005,Y -147.092,Z 1457.213,A 0.000,B 0.000,C 90.000,E1 218.338} C_DIS
LIN {X -0.001,Y -145.663,Z 1457.198,A 0.000,B 0.000,C 90.000,E1 215.598} C_DIS
LIN {X 0.002,Y -143.045,Z 1457.172,A 0.000,B 0.000,C 90.000,E1 211.003} C_DIS
LIN {X 0.003,Y -141.669,Z 1457.152,A 0.000,B 0.000,C 90.000,E1 207.308} C_DIS
LIN {X 0.047,Y -139.451,Z 1457.116,A 0.000,B 0.000,C 90.000,E1 200.791} C_DIS
LIN {X -0.032,Y -139.185,Z 1457.105,A 0.000,B 0.000,C 90.000,E1 198.960} C_DIS
LIN {X -0.009,Y -138.322,Z 1457.053,A 0.000,B 0.000,C 90.000,E1 189.613} C_DIS
LIN {X -0.002,Y -139.461,Z 1457.007,A 0.000,B 0.000,C 90.000,E1 181.203} C_DIS
LIN {X -0.062,Y -141.018,Z 1456.976,A 0.000,B 0.000,C 90.000,E1 175.641} C_DIS
LIN {X 0.028,Y -142.771,Z 1456.955,A 0.000,B 0.000,C 90.000,E1 171.894} C_DIS
LIN {X 0.015,Y -145.183,Z 1456.929,A 0.000,B 0.000,C 90.000,E1 167.285} C_DIS
LIN {X 0.017,Y -147.805,Z 1456.909,A 0.000,B 0.000,C 90.000,E1 163.614} C_DIS
LIN {X -0.089,Y -150.491,Z 1456.889,A 0.000,B 0.000,C 90.000,E1 160.007} C_DIS
LIN {X -0.016,Y -153.948,Z 1456.869,A 0.000,B 0.000,C 90.000,E1 156.357} C_DIS
LIN {X 0.048,Y -157.359,Z 1456.849,A 0.000,B 0.000,C 90.000,E1 152.743} C_DIS
LIN {X -0.010,Y -161.556,Z 1456.829,A 0.000,B 0.000,C 90.000,E1 149.203} C_DIS
LIN {X 0.002,Y -165.754,Z 1456.809,A 0.000,B 0.000,C 90.000,E1 145.674} C_DIS
LIN {X -0.010,Y -170.710,Z 1456.790,A 0.000,B 0.000,C 90.000,E1 142.190} C_DIS
LIN {X -0.099,Y -175.583,Z 1456.771,A 0.000,B 0.000,C 90.000,E1 138.771} C_DIS
LIN {X 0.019,Y -181.200,Z 1456.752,A 0.000,B 0.000,C 90.000,E1 135.324} C_DIS
LIN {X 0.013,Y -186.662,Z 1456.733,A 0.000,B 0.000,C 90.000,E1 131.962} C_DIS
LIN {X -0.043,Y -191.267,Z 1456.719,A 0.000,B 0.000,C 90.000,E1 129.483} C_DIS
LIN {X 0.037,Y -197.089,Z 1456.701,A 0.000,B 0.000,C 90.000,E1 126.171} C_DIS
LIN {X 0.062,Y -200.767,Z 1456.691,A 0.000,B 0.000,C 90.000,E1 124.326} C_DIS
LIN {X 0.062,Y -312.516,Z 1456.691,A 0.000,B 0.000,C 90.000,E1 124.326} C_DIS
LIN {X -0.132,Y -314.783,Z 1456.691,A 0.000,B 0.000,C 90.000,E1 124.326} C_DIS
LIN {X -0.096,Y -320.180,Z 1456.689,A 0.000,B 0.000,C 90.000,E1 124.040} C_DIS
LIN {X 0.211,Y -323.049,Z 1456.688,A 0.000,B 0.000,C 90.000,E1 123.706} C_DIS
LIN {X -0.095,Y -326.699,Z 1456.684,A 0.000,B 0.000,C 90.000,E1 123.214} C_DIS
LIN {X -0.004,Y -328.175,Z 1456.683,A 0.000,B 0.000,C 90.000,E1 122.880} C_DIS
LIN {X 0.162,Y -341.409,Z 1456.664,A 0.000,B 0.000,C 90.000,E1 119.411} C_DIS
LIN {X 0.096,Y -353.706,Z 1456.648,A 0.000,B 0.000,C 90.000,E1 116.668} C_DIS
LIN {X 0.216,Y -367.488,Z 1456.633,A 0.000,B 0.000,C 90.000,E1 113.951} C_DIS
LIN {X -0.029,Y -381.078,Z 1456.620,A 0.000,B 0.000,C 90.000,E1 111.642} C_DIS
LIN {X 0.133,Y -396.028,Z 1456.607,A 0.000,B 0.000,C 90.000,E1 109.322} C_DIS
LIN {X 0.038,Y -412.441,Z 1456.595,A 0.000,B 0.000,C 90.000,E1 107.094} C_DIS
LIN {X 0.116,Y -430.431,Z 1456.583,A 0.000,B 0.000,C 90.000,E1 104.898} C_DIS
LIN {X -0.193,Y -449.965,Z 1456.571,A 0.000,B 0.000,C 90.000,E1 102.827} C_DIS
LIN {X 0.108,Y -470.213,Z 1456.560,A 0.000,B 0.000,C 90.000,E1 100.838} C_DIS
LIN {X 0.083,Y -488.227,Z 1456.552,A 0.000,B 0.000,C 90.000,E1 99.265} C_DIS
LIN {X 0.238,Y -490.148,Z 1456.550,A 0.000,B 0.000,C 90.000,E1 99.029} C_DIS
LIN {X 0.063,Y -491.800,Z 1456.549,A 0.000,B 0.000,C 90.000,E1 98.803} C_DIS
LIN {X -0.039,Y -493.033,Z 1456.548,A 0.000,B 0.000,C 90.000,E1 98.568} C_DIS
LIN {X 0.194,Y -494.532,Z 1456.545,A 0.000,B 0.000,C 90.000,E1 98.049} C_DIS
LIN {X -0.054,Y -494.966,Z 1456.542,A 0.000,B 0.000,C 90.000,E1 97.587} C_DIS
LIN {X 0.198,Y -494.410,Z 1456.539,A 0.000,B 0.000,C 90.000,E1 97.068} C_DIS
LIN {X -0.038,Y -492.775,Z 1456.537,A 0.000,B 0.000,C 90.000,E1 96.606} C_DIS
LIN {X -0.130,Y -491.461,Z 1456.535,A 0.000,B 0.000,C 90.000,E1 96.372} C_DIS
LIN {X -0.126,Y -479.784,Z 1456.526,A 0.000,B 0.000,C 90.000,E1 94.645} C_DIS
LIN {X 0.083,Y -469.117,Z 1456.516,A 0.000,B 0.000,C 90.000,E1 92.865} C_DIS
LIN {X 0.023,Y -460.985,Z 1456.509,A 0.000,B 0.000,C 90.000,E1 91.604} C_DIS
LIN {X -0.177,Y -449.085,Z 1456.499,A 0.000,B 0.000,C 90.000,E1 89.828} C_DIS
LIN {X 0.185,Y -434.087,Z 1456.486,A 0.000,B 0.000,C 90.000,E1 87.421} C_DIS
LIN {X -0.076,Y -422.366,Z 1456.475,A 0.000,B 0.000,C 90.000,E1 85.584} C_DIS
LIN {X -0.111,Y -410.719,Z 1456.465,A 0.000,B 0.000,C 90.000,E1 83.685} C_DIS
LIN {X 0.022,Y -400.566,Z 1456.456,A 0.000,B 0.000,C 90.000,E1 82.008} C_DIS
LIN {X 0.084,Y -386.914,Z 1456.443,A 0.000,B 0.000,C 90.000,E1 79.746} C_DIS
LIN {X -0.041,Y -373.519,Z 1456.430,A 0.000,B 0.000,C 90.000,E1 77.465} C_DIS
LIN {X 0.049,Y -360.555,Z 1456.417,A 0.000,B 0.000,C 90.000,E1 75.102} C_DIS
LIN {X -0.045,Y -350.882,Z 1456.407,A 0.000,B 0.000,C 90.000,E1 73.323} C_DIS
LIN {X 0.113,Y -337.857,Z 1456.394,A 0.000,B 0.000,C 90.000,E1 70.859} C_DIS
LIN {X -0.141,Y -325.043,Z 1456.380,A 0.000,B 0.000,C 90.000,E1 68.411} C_DIS
LIN {X -0.103,Y -311.385,Z 1456.364,A 0.000,B 0.000,C 90.000,E1 65.537} C_DIS
LIN {X 0.104,Y -297.224,Z 1456.346,A 0.000,B 0.000,C 90.000,E1 62.231} C_DIS
LIN {X 0.160,Y -284.239,Z 1456.327,A 0.000,B 0.000,C 90.000,E1 58.869} C_DIS
LIN {X 0.085,Y -273.292,Z 1456.310,A 0.000,B 0.000,C 90.000,E1 55.801} C_DIS
LIN {X 0.015,Y -261.707,Z 1456.291,A 0.000,B 0.000,C 90.000,E1 52.316} C_DIS
LIN {X -0.105,Y -251.085,Z 1456.271,A 0.000,B 0.000,C 90.000,E1 48.771} C_DIS
LIN {X 0.094,Y -241.405,Z 1456.251,A 0.000,B 0.000,C 90.000,E1 45.081} C_DIS
LIN {X -0.004,Y -232.637,Z 1456.230,A 0.000,B 0.000,C 90.000,E1 41.391} C_DIS
LIN {X 0.028,Y -224.829,Z 1456.209,A 0.000,B 0.000,C 90.000,E1 37.604} C_DIS
LIN {X -0.055,Y -217.841,Z 1456.188,A 0.000,B 0.000,C 90.000,E1 33.785} C_DIS
LIN {X 0.010,Y -211.633,Z 1456.166,A 0.000,B 0.000,C 90.000,E1 29.873} C_DIS
LIN {X 0.019,Y -206.275,Z 1456.144,A 0.000,B 0.000,C 90.000,E1 25.924} C_DIS
LIN {X -0.040,Y -201.730,Z 1456.122,A 0.000,B 0.000,C 90.000,E1 21.950} C_DIS
LIN {X 0.020,Y -197.255,Z 1456.095,A 0.000,B 0.000,C 90.000,E1 17.094} C_DIS
LIN {X -0.093,Y -193.899,Z 1456.068,A 0.000,B 0.000,C 90.000,E1 12.243} C_DIS
LIN {X 0.007,Y -191.564,Z 1456.041,A 0.000,B 0.000,C 90.000,E1 7.296} C_DIS
LIN {X -0.051,Y -189.923,Z 1456.009,A 0.000,B 0.000,C 90.000,E1 1.547} C_DIS
LIN {X 0.030,Y -189.417,Z 1455.979,A 0.000,B 0.000,C 90.000,E1 356.216} C_DIS
LIN {X -0.014,Y -189.992,Z 1455.947,A 0.000,B 0.000,C 90.000,E1 350.443} C_DIS
LIN {X -0.026,Y -192.264,Z 1455.910,A 0.000,B 0.000,C 90.000,E1 343.850} C_DIS
LIN {X 0.069,Y -195.332,Z 1455.883,A 0.000,B 0.000,C 90.000,E1 338.901} C_DIS
LIN {X 0.010,Y -198.825,Z 1455.860,A 0.000,B 0.000,C 90.000,E1 334.845} C_DIS
LIN {X 0.043,Y -203.461,Z 1455.838,A 0.000,B 0.000,C 90.000,E1 330.795} C_DIS
LIN {X 0.087,Y -208.036,Z 1455.820,A 0.000,B 0.000,C 90.000,E1 327.582} C_DIS
LIN {X 0.126,Y -213.487,Z 1455.802,A 0.000,B 0.000,C 90.000,E1 324.402} C_DIS
LIN {X 0.036,Y -219.867,Z 1455.785,A 0.000,B 0.000,C 90.000,E1 321.295} C_DIS
LIN {X -0.019,Y -228.112,Z 1455.766,A 0.000,B 0.000,C 90.000,E1 317.838} C_DIS
LIN {X -0.017,Y -237.632,Z 1455.747,A 0.000,B 0.000,C 90.000,E1 314.433} C_DIS
LIN {X -0.052,Y -247.104,Z 1455.730,A 0.000,B 0.000,C 90.000,E1 311.472} C_DIS
LIN {X 0.023,Y -257.821,Z 1455.714,A 0.000,B 0.000,C 90.000,E1 308.543} C_DIS
LIN {X -0.116,Y -269.793,Z 1455.698,A 0.000,B 0.000,C 90.000,E1 305.724} C_DIS
LIN {X 0.136,Y -279.987,Z 1455.687,A 0.000,B 0.000,C 90.000,E1 303.579} C_DIS
LIN {X 0.081,Y -289.498,Z 1455.677,A 0.000,B 0.000,C 90.000,E1 301.878} C_DIS
LIN {X 0.017,Y -300.022,Z 1455.668,A 0.000,B 0.000,C 90.000,E1 300.207} C_DIS
LIN {X 0.085,Y -309.328,Z 1455.661,A 0.000,B 0.000,C 90.000,E1 298.871} C_DIS
LIN {X -0.028,Y -319.833,Z 1455.653,A 0.000,B 0.000,C 90.000,E1 297.590} C_DIS
LIN {X -0.058,Y -336.136,Z 1455.643,A 0.000,B 0.000,C 90.000,E1 295.796} C_DIS
LIN {X 0.058,Y -349.849,Z 1455.635,A 0.000,B 0.000,C 90.000,E1 294.387} C_DIS
LIN {X -0.034,Y -363.502,Z 1455.628,A 0.000,B 0.000,C 90.000,E1 293.025} C_DIS
LIN {X 0.186,Y -374.078,Z 1455.622,A 0.000,B 0.000,C 90.000,E1 291.897} C_DIS
LIN {X -0.010,Y -386.899,Z 1455.614,A 0.000,B 0.000,C 90.000,E1 290.556} C_DIS
LIN {X -0.113,Y -397.074,Z 1455.608,A 0.000,B 0.000,C 90.000,E1 289.450} C_DIS
LIN {X -0.155,Y -409.435,Z 1455.600,A 0.000,B 0.000,C 90.000,E1 288.055} C_DIS
LIN {X -0.128,Y -416.536,Z 1455.596,A 0.000,B 0.000,C 90.000,E1 287.221} C_DIS
LIN {X -0.039,Y -423.107,Z 1455.591,A 0.000,B 0.000,C 90.000,E1 286.386} C_DIS
LIN {X 0.122,Y -428.957,Z 1455.587,A 0.000,B 0.000,C 90.000,E1 285.552} C_DIS
LIN {X -0.086,Y -433.943,Z 1455.582,A 0.000,B 0.000,C 90.000,E1 284.773} C_DIS
LIN {X 0.065,Y -437.943,Z 1455.578,A 0.000,B 0.000,C 90.000,E1 283.953} C_DIS
LIN {X -0.071,Y -441.231,Z 1455.573,A 0.000,B 0.000,C 90.000,E1 283.175} C_DIS
LIN {X -0.072,Y -443.012,Z 1455.570,A 0.000,B 0.000,C 90.000,E1 282.647} C_DIS
LIN {X -0.067,Y -444.483,Z 1455.567,A 0.000,B 0.000,C 90.000,E1 282.119} C_DIS
LIN {X -0.050,Y -445.566,Z 1455.564,A 0.000,B 0.000,C 90.000,E1 281.591} C_DIS
LIN {X -0.112,Y -446.238,Z 1455.561,A 0.000,B 0.000,C 90.000,E1 281.074} C_DIS
LIN {X -0.080,Y -446.457,Z 1455.558,A 0.000,B 0.000,C 90.000,E1 280.546} C_DIS
LIN {X -0.047,Y -446.201,Z 1455.556,A 0.000,B 0.000,C 90.000,E1 280.018} C_DIS
LIN {X -0.089,Y -445.411,Z 1455.553,A 0.000,B 0.000,C 90.000,E1 279.500} C_DIS
LIN {X -0.060,Y -444.036,Z 1455.550,A 0.000,B 0.000,C 90.000,E1 278.973} C_DIS
LIN {X -0.104,Y -442.026,Z 1455.547,A 0.000,B 0.000,C 90.000,E1 278.454} C_DIS
LIN {X -0.153,Y -439.279,Z 1455.544,A 0.000,B 0.000,C 90.000,E1 277.936} C_DIS
LIN {X -0.161,Y -435.641,Z 1455.541,A 0.000,B 0.000,C 90.000,E1 277.409} C_DIS
LIN {X -0.016,Y -433.381,Z 1455.540,A 0.000,B 0.000,C 90.000,E1 277.125} C_DIS
LIN {X -0.064,Y -428.065,Z 1455.537,A 0.000,B 0.000,C 90.000,E1 276.606} C_DIS
LIN {X 0.166,Y -424.933,Z 1455.535,A 0.000,B 0.000,C 90.000,E1 276.315} C_DIS
LIN {X -0.183,Y -418.573,Z 1455.533,A 0.000,B 0.000,C 90.000,E1 275.910} C_DIS
LIN {X -0.169,Y -412.021,Z 1455.531,A 0.000,B 0.000,C 90.000,E1 275.511} C_DIS
LIN {X -0.007,Y -402.307,Z 1455.528,A 0.000,B 0.000,C 90.000,E1 274.992} C_DIS
LIN {X -0.188,Y -392.447,Z 1455.525,A 0.000,B 0.000,C 90.000,E1 274.588} C_DIS
LIN {X -0.083,Y -379.436,Z 1455.523,A 0.000,B 0.000,C 90.000,E1 274.073} C_DIS
LIN {X -0.081,Y -363.912,Z 1455.519,A 0.000,B 0.000,C 90.000,E1 273.498} C_DIS
LIN {X -0.020,Y -353.846,Z 1455.517,A 0.000,B 0.000,C 90.000,E1 273.154} C_DIS
LIN {X 0.026,Y -343.537,Z 1455.516,A 0.000,B 0.000,C 90.000,E1 272.865} C_DIS
LIN {X 0.080,Y -336.947,Z 1455.515,A 0.000,B 0.000,C 90.000,E1 272.694} C_DIS
LIN {X -0.130,Y -325.733,Z 1455.514,A 0.000,B 0.000,C 90.000,E1 272.522} C_DIS
LIN {X -0.113,Y -312.890,Z 1455.513,A 0.000,B 0.000,C 90.000,E1 272.350} C_DIS
LIN {X -0.013,Y -300.158,Z 1455.512,A 0.000,B 0.000,C 90.000,E1 272.236} C_DIS
LIN {X -0.043,Y -181.227,Z 1455.512,A 0.000,B 0.000,C 90.000,E1 272.236} C_DIS
LIN {X -0.035,Y -181.564,Z 1455.503,A 0.000,B 0.000,C 90.000,E1 270.516} C_DIS
LIN {X -0.045,Y -181.121,Z 1455.489,A 0.000,B 0.000,C 90.000,E1 267.993} C_DIS
LIN {X -0.056,Y -180.907,Z 1455.475,A 0.000,B 0.000,C 90.000,E1 265.469} C_DIS
LIN {X 0.000,Y -180.729,Z 1455.470,A 0.000,B 0.000,C 90.000,E1 264.609} C_DIS
LIN {X 0.098,Y -178.817,Z 1455.442,A 0.000,B 0.000,C 90.000,E1 259.511} C_DIS
LIN {X 0.004,Y -175.862,Z 1455.414,A 0.000,B 0.000,C 90.000,E1 254.448} C_DIS
LIN {X 0.053,Y -173.828,Z 1455.399,A 0.000,B 0.000,C 90.000,E1 251.873} C_DIS
LIN {X -0.012,Y -171.496,Z 1455.380,A 0.000,B 0.000,C 90.000,E1 248.465} C_DIS
LIN {X -0.024,Y -167.724,Z 1455.356,A 0.000,B 0.000,C 90.000,E1 244.152} C_DIS
LIN {X -0.009,Y -166.418,Z 1455.347,A 0.000,B 0.000,C 90.000,E1 242.410} C_DIS
LIN {X -0.010,Y -163.140,Z 1455.327,A 0.000,B 0.000,C 90.000,E1 238.918} C_DIS
LIN {X -0.044,Y -161.094,Z 1455.313,A 0.000,B 0.000,C 90.000,E1 236.294} C_DIS
LIN {X -0.060,Y -157.823,Z 1455.293,A 0.000,B 0.000,C 90.000,E1 232.763} C_DIS
LIN {X 0.003,Y -155.857,Z 1455.278,A 0.000,B 0.000,C 90.000,E1 230.070} C_DIS
LIN {X 0.058,Y -152.107,Z 1455.253,A 0.000,B 0.000,C 90.000,E1 225.567} C_DIS
LIN {X 0.077,Y -150.357,Z 1455.238,A 0.000,B 0.000,C 90.000,E1 222.852} C_DIS
LIN {X 0.005,Y -147.093,Z 1455.213,A 0.000,B 0.000,C 90.000,E1 218.338} C_DIS
LIN {X 0.000,Y -145.663,Z 1455.198,A 0.000,B 0.000,C 90.000,E1 215.598} C_DIS
LIN {X 0.003,Y -143.045,Z 1455.172,A 0.000,B 0.000,C 90.000,E1 211.003} C_DIS
LIN {X 0.004,Y -141.669,Z 1455.152,A 0.000,B 0.000,C 90.000,E1 207.308} C_DIS
LIN {X 0.048,Y -139.452,Z 1455.116,A 0.000,B 0.000,C 90.000,E1 200.791} C_DIS
LIN {X -0.031,Y -139.186,Z 1455.105,A 0.000,B 0.000,C 90.000,E1 198.960} C_DIS
LIN {X -0.008,Y -138.322,Z 1455.053,A 0.000,B 0.000,C 90.000,E1 189.613} C_DIS
LIN {X -0.001,Y -139.461,Z 1455.007,A 0.000,B 0.000,C 90.000,E1 181.203} C_DIS
LIN {X -0.061,Y -141.018,Z 1454.976,A 0.000,B 0.000,C 90.000,E1 175.641} C_DIS
LIN {X 0.029,Y -142.771,Z 1454.955,A 0.000,B 0.000,C 90.000,E1 171.894} C_DIS
LIN {X -0.016,Y -145.183,Z 1454.929,A 0.000,B 0.000,C 90.000,E1 167.297} C_DIS
LIN {X 0.018,Y -147.804,Z 1454.909,A 0.000,B 0.000,C 90.000,E1 163.614} C_DIS
LIN {X -0.087,Y -150.490,Z 1454.889,A 0.000,B 0.000,C 90.000,E1 160.007} C_DIS
LIN {X -0.014,Y -153.947,Z 1454.869,A 0.000,B 0.000,C 90.000,E1 156.357} C_DIS
LIN {X 0.049,Y -157.359,Z 1454.849,A 0.000,B 0.000,C 90.000,E1 152.743} C_DIS
LIN {X -0.009,Y -161.556,Z 1454.829,A 0.000,B 0.000,C 90.000,E1 149.203} C_DIS
LIN {X 0.003,Y -165.754,Z 1454.809,A 0.000,B 0.000,C 90.000,E1 145.674} C_DIS
LIN {X -0.010,Y -170.709,Z 1454.790,A 0.000,B 0.000,C 90.000,E1 142.190} C_DIS
LIN {X -0.098,Y -175.582,Z 1454.771,A 0.000,B 0.000,C 90.000,E1 138.771} C_DIS
LIN {X 0.021,Y -181.200,Z 1454.752,A 0.000,B 0.000,C 90.000,E1 135.324} C_DIS
LIN {X 0.014,Y -186.662,Z 1454.733,A 0.000,B 0.000,C 90.000,E1 131.962} C_DIS
LIN {X -0.043,Y -191.266,Z 1454.719,A 0.000,B 0.000,C 90.000,E1 129.483} C_DIS
LIN {X 0.038,Y -197.087,Z 1454.701,A 0.000,B 0.000,C 90.000,E1 126.171} C_DIS
LIN {X -0.115,Y -200.714,Z 1454.691,A 0.000,B 0.000,C 90.000,E1 124.405} C_DIS
LIN {X 0.029,Y -312.445,Z 1454.691,A 0.000,B 0.000,C 90.000,E1 124.358} C_DIS
LIN {X 0.054,Y -317.684,Z 1454.690,A 0.000,B 0.000,C 90.000,E1 124.199} C_DIS
LIN {X 0.078,Y -320.016,Z 1454.689,A 0.000,B 0.000,C 90.000,E1 124.040} C_DIS
LIN {X 0.213,Y -323.158,Z 1454.688,A 0.000,B 0.000,C 90.000,E1 123.706} C_DIS
LIN {X 0.149,Y -326.750,Z 1454.684,A 0.000,B 0.000,C 90.000,E1 123.166} C_DIS
LIN {X -0.032,Y -328.188,Z 1454.683,A 0.000,B 0.000,C 90.000,E1 122.880} C_DIS
LIN {X -0.011,Y -340.126,Z 1454.665,A 0.000,B 0.000,C 90.000,E1 119.745} C_DIS
LIN {X -0.120,Y -352.270,Z 1454.650,A 0.000,B 0.000,C 90.000,E1 117.001} C_DIS
LIN {X 0.114,Y -365.881,Z 1454.635,A 0.000,B 0.000,C 90.000,E1 114.259} C_DIS
LIN {X 0.176,Y -379.310,Z 1454.622,A 0.000,B 0.000,C 90.000,E1 111.897} C_DIS
LIN {X -0.065,Y -394.087,Z 1454.609,A 0.000,B 0.000,C 90.000,E1 109.631} C_DIS
LIN {X -0.211,Y -410.313,Z 1454.597,A 0.000,B 0.000,C 90.000,E1 107.402} C_DIS
LIN {X -0.078,Y -428.102,Z 1454.584,A 0.000,B 0.000,C 90.000,E1 105.190} C_DIS
LIN {X -0.064,Y -447.478,Z 1454.573,A 0.000,B 0.000,C 90.000,E1 103.063} C_DIS
LIN {X 0.073,Y -467.657,Z 1454.562,A 0.000,B 0.000,C 90.000,E1 101.074} C_DIS
LIN {X 0.048,Y -488.226,Z 1454.552,A 0.000,B 0.000,C 90.000,E1 99.265} C_DIS
LIN {X 0.203,Y -490.121,Z 1454.550,A 0.000,B 0.000,C 90.000,E1 99.029} C_DIS
LIN {X 0.026,Y -491.752,Z 1454.549,A 0.000,B 0.000,C 90.000,E1 98.803} C_DIS
LIN {X -0.075,Y -492.970,Z 1454.548,A 0.000,B 0.000,C 90.000,E1 98.568} C_DIS
LIN {X 0.158,Y -494.445,Z 1454.545,A 0.000,B 0.000,C 90.000,E1 98.049} C_DIS
LIN {X -0.090,Y -494.858,Z 1454.542,A 0.000,B 0.000,C 90.000,E1 97.587} C_DIS
LIN {X 0.161,Y -494.281,Z 1454.539,A 0.000,B 0.000,C 90.000,E1 97.068} C_DIS
LIN {X -0.076,Y -492.622,Z 1454.537,A 0.000,B 0.000,C 90.000,E1 96.606} C_DIS
LIN {X -0.168,Y -491.292,Z 1454.535,A 0.000,B 0.000,C 90.000,E1 96.372} C_DIS
LIN {X -0.166,Y -479.625,Z 1454.526,A 0.000,B 0.000,C 90.000,E1 94.645} C_DIS
LIN {X 0.041,Y -468.945,Z 1454.516,A 0.000,B 0.000,C 90.000,E1 92.865} C_DIS
LIN {X -0.021,Y -460.773,Z 1454.509,A 0.000,B 0.000,C 90.000,E1 91.604} C_DIS
LIN {X -0.224,Y -448.863,Z 1454.499,A 0.000,B 0.000,C 90.000,E1 89.828} C_DIS
LIN {X 0.134,Y -433.909,Z 1454.486,A 0.000,B 0.000,C 90.000,E1 87.421} C_DIS
LIN {X -0.129,Y -422.241,Z 1454.475,A 0.000,B 0.000,C 90.000,E1 85.584} C_DIS
LIN {X -0.164,Y -410.615,Z 1454.465,A 0.000,B 0.000,C 90.000,E1 83.685} C_DIS
LIN {X -0.032,Y -400.508,Z 1454.456,A 0.000,B 0.000,C 90.000,E1 82.008} C_DIS
LIN {X 0.031,Y -386.887,Z 1454.443,A 0.000,B 0.000,C 90.000,E1 79.746} C_DIS
LIN {X -0.093,Y -373.525,Z 1454.430,A 0.000,B 0.000,C 90.000,E1 77.465} C_DIS
LIN {X -0.001,Y -360.533,Z 1454.417,A 0.000,B 0.000,C 90.000,E1 75.102} C_DIS
LIN {X -0.095,Y -350.847,Z 1454.407,A 0.000,B 0.000,C 90.000,E1 73.323} C_DIS
LIN {X 0.060,Y -339.465,Z 1454.395,A 0.000,B 0.000,C 90.000,E1 71.167} C_DIS
LIN {X -0.157,Y -326.580,Z 1454.382,A 0.000,B 0.000,C 90.000,E1 68.720} C_DIS
LIN {X -0.073,Y -312.792,Z 1454.366,A 0.000,B 0.000,C 90.000,E1 65.845} C_DIS
LIN {X 0.045,Y -298.498,Z 1454.348,A 0.000,B 0.000,C 90.000,E1 62.564} C_DIS
LIN {X 0.138,Y -285.407,Z 1454.329,A 0.000,B 0.000,C 90.000,E1 59.203} C_DIS
LIN {X -0.059,Y -274.454,Z 1454.312,A 0.000,B 0.000,C 90.000,E1 56.167} C_DIS
LIN {X 0.115,Y -262.842,Z 1454.293,A 0.000,B 0.000,C 90.000,E1 52.637} C_DIS
LIN {X -0.018,Y -253.147,Z 1454.275,A 0.000,B 0.000,C 90.000,E1 49.461} C_DIS
LIN {X 0.075,Y -243.327,Z 1454.255,A 0.000,B 0.000,C 90.000,E1 45.810} C_DIS
LIN {X 0.021,Y -234.419,Z 1454.234,A 0.000,B 0.000,C 90.000,E1 42.123} C_DIS
LIN {X -0.076,Y -226.445,Z 1454.213,A 0.000,B 0.000,C 90.000,E1 38.382} C_DIS
LIN {X 0.016,Y -219.319,Z 1454.192,A 0.000,B 0.000,C 90.000,E1 34.532} C_DIS
LIN {X -0.060,Y -212.969,Z 1454.170,A 0.000,B 0.000,C 90.000,E1 30.669} C_DIS
LIN {X -0.096,Y -207.450,Z 1454.148,A 0.000,B 0.000,C 90.000,E1 26.744} C_DIS
LIN {X -0.115,Y -202.771,Z 1454.126,A 0.000,B 0.000,C 90.000,E1 22.770} C_DIS
LIN {X -0.066,Y -198.164,Z 1454.099,A 0.000,B 0.000,C 90.000,E1 17.928} C_DIS
LIN {X -0.101,Y -194.611,Z 1454.072,A 0.000,B 0.000,C 90.000,E1 13.063} C_DIS
LIN {X 0.059,Y -192.179,Z 1454.045,A 0.000,B 0.000,C 90.000,E1 8.106} C_DIS
LIN {X 0.045,Y -190.349,Z 1454.013,A 0.000,B 0.000,C 90.000,E1 2.350} C_DIS
LIN {X 0.003,Y -189.747,Z 1453.988,A 0.000,B 0.000,C 90.000,E1 357.879} C_DIS
LIN {X 0.080,Y -189.933,Z 1453.956,A 0.000,B 0.000,C 90.000,E1 352.072} C_DIS
LIN {X -0.108,Y -191.396,Z 1453.924,A 0.000,B 0.000,C 90.000,E1 346.353} C_DIS
LIN {X 0.060,Y -194.349,Z 1453.892,A 0.000,B 0.000,C 90.000,E1 340.550} C_DIS
LIN {X 0.022,Y -198.194,Z 1453.865,A 0.000,B 0.000,C 90.000,E1 335.665} C_DIS
LIN {X -0.055,Y -202.582,Z 1453.842,A 0.000,B 0.000,C 90.000,E1 331.641} C_DIS
LIN {X 0.028,Y -208.178,Z 1453.820,A 0.000,B 0.000,C 90.000,E1 327.612} C_DIS
LIN {X -0.113,Y -213.619,Z 1453.802,A 0.000,B 0.000,C 90.000,E1 324.482} C_DIS
LIN {X -0.039,Y -220.012,Z 1453.785,A 0.000,B 0.000,C 90.000,E1 321.331} C_DIS
LIN {X 0.051,Y -228.271,Z 1453.766,A 0.000,B 0.000,C 90.000,E1 317.838} C_DIS
LIN {X 0.060,Y -237.784,Z 1453.747,A 0.000,B 0.000,C 90.000,E1 314.433} C_DIS
LIN {X 0.041,Y -246.010,Z 1453.733,A 0.000,B 0.000,C 90.000,E1 311.838} C_DIS
LIN {X 0.087,Y -256.569,Z 1453.716,A 0.000,B 0.000,C 90.000,E1 308.910} C_DIS
LIN {X -0.078,Y -268.348,Z 1453.700,A 0.000,B 0.000,C 90.000,E1 306.091} C_DIS
LIN {X -0.019,Y -276.582,Z 1453.691,A 0.000,B 0.000,C 90.000,E1 304.326} C_DIS
LIN {X -0.136,Y -285.631,Z 1453.681,A 0.000,B 0.000,C 90.000,E1 302.625} C_DIS
LIN {X -0.117,Y -295.745,Z 1453.672,A 0.000,B 0.000,C 90.000,E1 300.924} C_DIS
LIN {X 0.156,Y -304.589,Z 1453.664,A 0.000,B 0.000,C 90.000,E1 299.539} C_DIS
LIN {X 0.096,Y -311.867,Z 1453.659,A 0.000,B 0.000,C 90.000,E1 298.565} C_DIS
LIN {X -0.096,Y -322.362,Z 1453.652,A 0.000,B 0.000,C 90.000,E1 297.334} C_DIS
LIN {X -0.097,Y -335.908,Z 1453.644,A 0.000,B 0.000,C 90.000,E1 295.848} C_DIS
LIN {X 0.065,Y -352.335,Z 1453.634,A 0.000,B 0.000,C 90.000,E1 294.155} C_DIS
LIN {X -0.146,Y -365.842,Z 1453.627,A 0.000,B 0.000,C 90.000,E1 292.823} C_DIS
LIN {X -0.057,Y -376.290,Z 1453.621,A 0.000,B 0.000,C 90.000,E1 291.716} C_DIS
LIN {X -0.122,Y -386.706,Z 1453.614,A 0.000,B 0.000,C 90.000,E1 290.610} C_DIS
LIN {X 0.123,Y -396.899,Z 1453.608,A 0.000,B 0.000,C 90.000,E1 289.450} C_DIS
LIN {X 0.049,Y -409.330,Z 1453.600,A 0.000,B 0.000,C 90.000,E1 288.055} C_DIS
LIN {X 0.077,Y -416.464,Z 1453.596,A 0.000,B 0.000,C 90.000,E1 287.221} C_DIS
LIN {X 0.169,Y -423.083,Z 1453.591,A 0.000,B 0.000,C 90.000,E1 286.386} C_DIS
LIN {X 0.172,Y -427.137,Z 1453.588,A 0.000,B 0.000,C 90.000,E1 285.843} C_DIS
LIN {X -0.048,Y -432.430,Z 1453.584,A 0.000,B 0.000,C 90.000,E1 285.064} C_DIS
LIN {X 0.082,Y -436.807,Z 1453.579,A 0.000,B 0.000,C 90.000,E1 284.245} C_DIS
LIN {X 0.055,Y -439.251,Z 1453.576,A 0.000,B 0.000,C 90.000,E1 283.716} C_DIS
LIN {X 0.147,Y -441.389,Z 1453.573,A 0.000,B 0.000,C 90.000,E1 283.175} C_DIS
LIN {X 0.149,Y -443.190,Z 1453.570,A 0.000,B 0.000,C 90.000,E1 282.647} C_DIS
LIN {X 0.157,Y -444.671,Z 1453.567,A 0.000,B 0.000,C 90.000,E1 282.119} C_DIS
LIN {X 0.174,Y -445.799,Z 1453.565,A 0.000,B 0.000,C 90.000,E1 281.591} C_DIS
LIN {X 0.113,Y -446.530,Z 1453.562,A 0.000,B 0.000,C 90.000,E1 281.074} C_DIS
LIN {X 0.147,Y -446.773,Z 1453.559,A 0.000,B 0.000,C 90.000,E1 280.546} C_DIS
LIN {X 0.181,Y -446.568,Z 1453.556,A 0.000,B 0.000,C 90.000,E1 280.018} C_DIS
LIN {X 0.140,Y -445.819,Z 1453.553,A 0.000,B 0.000,C 90.000,E1 279.500} C_DIS
LIN {X 0.172,Y -444.514,Z 1453.550,A 0.000,B 0.000,C 90.000,E1 278.973} C_DIS
LIN {X 0.130,Y -442.585,Z 1453.547,A 0.000,B 0.000,C 90.000,E1 278.454} C_DIS
LIN {X -0.082,Y -441.359,Z 1453.546,A 0.000,B 0.000,C 90.000,E1 278.219} C_DIS
LIN {X -0.138,Y -438.276,Z 1453.543,A 0.000,B 0.000,C 90.000,E1 277.701} C_DIS
LIN {X -0.209,Y -434.194,Z 1453.540,A 0.000,B 0.000,C 90.000,E1 277.182} C_DIS
LIN {X 0.132,Y -428.927,Z 1453.537,A 0.000,B 0.000,C 90.000,E1 276.606} C_DIS
LIN {X -0.103,Y -425.817,Z 1453.535,A 0.000,B 0.000,C 90.000,E1 276.372} C_DIS
LIN {X -0.097,Y -419.486,Z 1453.533,A 0.000,B 0.000,C 90.000,E1 275.910} C_DIS
LIN {X -0.095,Y -412.957,Z 1453.531,A 0.000,B 0.000,C 90.000,E1 275.511} C_DIS
LIN {X -0.071,Y -406.478,Z 1453.529,A 0.000,B 0.000,C 90.000,E1 275.163} C_DIS
LIN {X -0.010,Y -396.653,Z 1453.526,A 0.000,B 0.000,C 90.000,E1 274.702} C_DIS
LIN {X 0.023,Y -386.923,Z 1453.524,A 0.000,B 0.000,C 90.000,E1 274.302} C_DIS
LIN {X -0.010,Y -368.238,Z 1453.520,A 0.000,B 0.000,C 90.000,E1 273.612} C_DIS
LIN {X 0.002,Y -358.456,Z 1453.518,A 0.000,B 0.000,C 90.000,E1 273.269} C_DIS
LIN {X -0.098,Y -348.060,Z 1453.516,A 0.000,B 0.000,C 90.000,E1 272.980} C_DIS
LIN {X 0.104,Y -337.889,Z 1453.515,A 0.000,B 0.000,C 90.000,E1 272.694} C_DIS
LIN {X -0.139,Y -326.522,Z 1453.514,A 0.000,B 0.000,C 90.000,E1 272.522} C_DIS
LIN {X -0.112,Y -313.688,Z 1453.513,A 0.000,B 0.000,C 90.000,E1 272.350} C_DIS
LIN {X -0.003,Y -301.764,Z 1453.512,A 0.000,B 0.000,C 90.000,E1 272.236} C_DIS
LIN {X -0.036,Y -181.227,Z 1453.512,A 0.000,B 0.000,C 90.000,E1 272.236} C_DIS
LIN {X -0.024,Y -181.564,Z 1453.503,A 0.000,B 0.000,C 90.000,E1 270.516} C_DIS
LIN {X -0.034,Y -181.121,Z 1453.489,A 0.000,B 0.000,C 90.000,E1 267.993} C_DIS
LIN {X -0.046,Y -180.907,Z 1453.475,A 0.000,B 0.000,C 90.000,E1 265.469} C_DIS
LIN {X 0.011,Y -180.729,Z 1453.470,A 0.000,B 0.000,C 90.000,E1 264.609} C_DIS
LIN {X -0.068,Y -178.819,Z 1453.442,A 0.000,B 0.000,C 90.000,E1 259.567} C_DIS
LIN {X 0.015,Y -175.864,Z 1453.414,A 0.000,B 0.000,C 90.000,E1 254.448} C_DIS
LIN {X 0.064,Y -173.831,Z 1453.399,A 0.000,B 0.000,C 90.000,E1 251.873} C_DIS
LIN {X -0.001,Y -171.499,Z 1453.380,A 0.000,B 0.000,C 90.000,E1 248.465} C_DIS
LIN {X -0.014,Y -167.726,Z 1453.356,A 0.000,B 0.000,C 90.000,E1 244.152} C_DIS
LIN {X 0.002,Y -166.421,Z 1453.347,A 0.000,B 0.000,C 90.000,E1 242.410} C_DIS
LIN {X 0.000,Y -163.143,Z 1453.327,A 0.000,B 0.000,C 90.000,E1 238.918} C_DIS
LIN {X -0.035,Y -161.097,Z 1453.313,A 0.000,B 0.000,C 90.000,E1 236.294} C_DIS
LIN {X -0.051,Y -157.826,Z 1453.293,A 0.000,B 0.000,C 90.000,E1 232.763} C_DIS
LIN {X 0.013,Y -155.859,Z 1453.278,A 0.000,B 0.000,C 90.000,E1 230.070} C_DIS
LIN {X 0.068,Y -152.110,Z 1453.253,A 0.000,B 0.000,C 90.000,E1 225.567} C_DIS
LIN {X -0.024,Y -150.360,Z 1453.238,A 0.000,B 0.000,C 90.000,E1 222.894} C_DIS
LIN {X 0.015,Y -147.095,Z 1453.213,A 0.000,B 0.000,C 90.000,E1 218.338} C_DIS
LIN {X 0.010,Y -145.665,Z 1453.198,A 0.000,B 0.000,C 90.000,E1 215.598} C_DIS
LIN {X 0.012,Y -143.047,Z 1453.172,A 0.000,B 0.000,C 90.000,E1 211.003} C_DIS
LIN {X 0.013,Y -141.671,Z 1453.152,A 0.000,B 0.000,C 90.000,E1 207.308} C_DIS
LIN {X 0.057,Y -139.452,Z 1453.116,A 0.000,B 0.000,C 90.000,E1 200.791} C_DIS
LIN {X -0.022,Y -139.187,Z 1453.105,A 0.000,B 0.000,C 90.000,E1 198.960} C_DIS
LIN {X 0.001,Y -138.323,Z 1453.053,A 0.000,B 0.000,C 90.000,E1 189.613} C_DIS
LIN {X 0.008,Y -139.460,Z 1453.007,A 0.000,B 0.000,C 90.000,E1 181.203} C_DIS
LIN {X -0.052,Y -141.016,Z 1452.976,A 0.000,B 0.000,C 90.000,E1 175.641} C_DIS
LIN {X 0.039,Y -142.770,Z 1452.955,A 0.000,B 0.000,C 90.000,E1 171.894} C_DIS
LIN {X -0.006,Y -145.180,Z 1452.929,A 0.000,B 0.000,C 90.000,E1 167.297} C_DIS
LIN {X 0.027,Y -147.802,Z 1452.909,A 0.000,B 0.000,C 90.000,E1 163.614} C_DIS
LIN {X -0.078,Y -150.488,Z 1452.889,A 0.000,B 0.000,C 90.000,E1 160.007} C_DIS
LIN {X -0.005,Y -153.943,Z 1452.869,A 0.000,B 0.000,C 90.000,E1 156.357} C_DIS
LIN {X 0.058,Y -157.355,Z 1452.849,A 0.000,B 0.000,C 90.000,E1 152.743} C_DIS
LIN {X 0.001,Y -161.551,Z 1452.829,A 0.000,B 0.000,C 90.000,E1 149.203} C_DIS
LIN {X 0.014,Y -165.749,Z 1452.809,A 0.000,B 0.000,C 90.000,E1 145.674} C_DIS
LIN {X 0.001,Y -170.703,Z 1452.790,A 0.000,B 0.000,C 90.000,E1 142.190} C_DIS
LIN {X -0.088,Y -175.577,Z 1452.771,A 0.000,B 0.000,C 90.000,E1 138.771} C_DIS
LIN {X 0.031,Y -181.195,Z 1452.752,A 0.000,B 0.000,C 90.000,E1 135.324} C_DIS
LIN {X 0.025,Y -186.656,Z 1452.733,A 0.000,B 0.000,C 90.000,E1 131.962} C_DIS
LIN {X -0.032,Y -191.261,Z 1452.719,A 0.000,B 0.000,C 90.000,E1 129.483} C_DIS
LIN {X 0.049,Y -197.082,Z 1452.701,A 0.000,B 0.000,C 90.000,E1 126.171} C_DIS
LIN {X -0.040,Y -200.674,Z 1452.691,A 0.000,B 0.000,C 90.000,E1 124.405} C_DIS
LIN {X -0.112,Y -312.799,Z 1452.691,A 0.000,B 0.000,C 90.000,E1 124.405} C_DIS
LIN {X 0.047,Y -313.994,Z 1452.691,A 0.000,B 0.000,C 90.000,E1 124.358} C_DIS
LIN {X 0.072,Y -317.961,Z 1452.690,A 0.000,B 0.000,C 90.000,E1 124.199} C_DIS
LIN {X -0.083,Y -320.178,Z 1452.689,A 0.000,B 0.000,C 90.000,E1 124.072} C_DIS
LIN {X -0.217,Y -323.231,Z 1452.688,A 0.000,B 0.000,C 90.000,E1 123.785} C_DIS
LIN {X 0.097,Y -326.813,Z 1452.684,A 0.000,B 0.000,C 90.000,E1 123.166} C_DIS
LIN {X -0.083,Y -328.214,Z 1452.683,A 0.000,B 0.000,C 90.000,E1 122.880} C_DIS
LIN {X -0.065,Y -340.141,Z 1452.665,A 0.000,B 0.000,C 90.000,E1 119.745} C_DIS
LIN {X -0.175,Y -352.290,Z 1452.650,A 0.000,B 0.000,C 90.000,E1 117.001} C_DIS
LIN {X 0.057,Y -365.905,Z 1452.635,A 0.000,B 0.000,C 90.000,E1 114.259} C_DIS
LIN {X 0.118,Y -379.339,Z 1452.622,A 0.000,B 0.000,C 90.000,E1 111.897} C_DIS
LIN {X -0.123,Y -394.120,Z 1452.609,A 0.000,B 0.000,C 90.000,E1 109.631} C_DIS
LIN {X 0.121,Y -410.352,Z 1452.596,A 0.000,B 0.000,C 90.000,E1 107.347} C_DIS
LIN {X -0.140,Y -428.146,Z 1452.584,A 0.000,B 0.000,C 90.000,E1 105.190} C_DIS
LIN {X -0.127,Y -447.527,Z 1452.573,A 0.000,B 0.000,C 90.000,E1 103.063} C_DIS
LIN {X 0.012,Y -467.708,Z 1452.562,A 0.000,B 0.000,C 90.000,E1 101.074} C_DIS
LIN {X -0.012,Y -488.252,Z 1452.552,A 0.000,B 0.000,C 90.000,E1 99.265} C_DIS
LIN {X 0.143,Y -490.115,Z 1452.550,A 0.000,B 0.000,C 90.000,E1 99.029} C_DIS
LIN {X -0.033,Y -491.721,Z 1452.549,A 0.000,B 0.000,C 90.000,E1 98.803} C_DIS
LIN {X -0.134,Y -492.921,Z 1452.547,A 0.000,B 0.000,C 90.000,E1 98.568} C_DIS
LIN {X 0.099,Y -494.364,Z 1452.545,A 0.000,B 0.000,C 90.000,E1 98.049} C_DIS
LIN {X -0.151,Y -494.751,Z 1452.542,A 0.000,B 0.000,C 90.000,E1 97.587} C_DIS
LIN {X 0.100,Y -494.148,Z 1452.539,A 0.000,B 0.000,C 90.000,E1 97.068} C_DIS
LIN {X -0.136,Y -492.458,Z 1452.537,A 0.000,B 0.000,C 90.000,E1 96.606} C_DIS
LIN {X -0.229,Y -491.108,Z 1452.535,A 0.000,B 0.000,C 90.000,E1 96.372} C_DIS
LIN {X -0.229,Y -479.413,Z 1452.526,A 0.000,B 0.000,C 90.000,E1 94.645} C_DIS
LIN {X -0.025,Y -468.744,Z 1452.516,A 0.000,B 0.000,C 90.000,E1 92.865} C_DIS
LIN {X -0.088,Y -460.539,Z 1452.509,A 0.000,B 0.000,C 90.000,E1 91.604} C_DIS
LIN {X -0.085,Y -446.939,Z 1452.497,A 0.000,B 0.000,C 90.000,E1 89.542} C_DIS
LIN {X 0.060,Y -433.711,Z 1452.486,A 0.000,B 0.000,C 90.000,E1 87.421} C_DIS
LIN {X -0.205,Y -422.095,Z 1452.475,A 0.000,B 0.000,C 90.000,E1 85.584} C_DIS
LIN {X 0.167,Y -410.504,Z 1452.465,A 0.000,B 0.000,C 90.000,E1 83.628} C_DIS
LIN {X -0.079,Y -398.716,Z 1452.454,A 0.000,B 0.000,C 90.000,E1 81.724} C_DIS
LIN {X -0.045,Y -386.834,Z 1452.443,A 0.000,B 0.000,C 90.000,E1 79.746} C_DIS
LIN {X -0.167,Y -373.503,Z 1452.430,A 0.000,B 0.000,C 90.000,E1 77.465} C_DIS
LIN {X -0.073,Y -360.521,Z 1452.417,A 0.000,B 0.000,C 90.000,E1 75.102} C_DIS
LIN {X -0.133,Y -349.199,Z 1452.406,A 0.000,B 0.000,C 90.000,E1 73.015} C_DIS
LIN {X -0.003,Y -337.795,Z 1452.394,A 0.000,B 0.000,C 90.000,E1 70.859} C_DIS
LIN {X 0.006,Y -323.394,Z 1452.378,A 0.000,B 0.000,C 90.000,E1 68.050} C_DIS
LIN {X 0.032,Y -308.300,Z 1452.360,A 0.000,B 0.000,C 90.000,E1 64.845} C_DIS
LIN {X -0.122,Y -293.011,Z 1452.340,A 0.000,B 0.000,C 90.000,E1 61.257} C_DIS
LIN {X -0.044,Y -280.395,Z 1452.321,A 0.000,B 0.000,C 90.000,E1 57.867} C_DIS
LIN {X -0.073,Y -269.682,Z 1452.304,A 0.000,B 0.000,C 90.000,E1 54.769} C_DIS
LIN {X -0.143,Y -259.515,Z 1452.287,A 0.000,B 0.000,C 90.000,E1 51.618} C_DIS
LIN {X 0.001,Y -249.135,Z 1452.267,A 0.000,B 0.000,C 90.000,E1 48.000} C_DIS
LIN {X -0.037,Y -239.732,Z 1452.246,A 0.000,B 0.000,C 90.000,E1 44.352} C_DIS
LIN {X -0.011,Y -231.213,Z 1452.226,A 0.000,B 0.000,C 90.000,E1 40.620} C_DIS
LIN {X 0.013,Y -223.620,Z 1452.205,A 0.000,B 0.000,C 90.000,E1 36.824} C_DIS
LIN {X 0.073,Y -216.811,Z 1452.183,A 0.000,B 0.000,C 90.000,E1 32.959} C_DIS
LIN {X -0.008,Y -210.808,Z 1452.161,A 0.000,B 0.000,C 90.000,E1 29.077} C_DIS
LIN {X -0.120,Y -205.646,Z 1452.140,A 0.000,B 0.000,C 90.000,E1 25.155} C_DIS
LIN {X 0.094,Y -201.314,Z 1452.117,A 0.000,B 0.000,C 90.000,E1 21.099} C_DIS
LIN {X 0.080,Y -197.073,Z 1452.090,A 0.000,B 0.000,C 90.000,E1 16.260} C_DIS
LIN {X -0.074,Y -193.563,Z 1452.059,A 0.000,B 0.000,C 90.000,E1 10.602} C_DIS
LIN {X -0.076,Y -191.517,Z 1452.031,A 0.000,B 0.000,C 90.000,E1 5.682} C_DIS
LIN {X 0.000,Y -190.238,Z 1452.000,A 0.000,B 0.000,C 90.000,E1 360.000} C_DIS
LIN {X 0.033,Y -190.028,Z 1451.965,A 0.000,B 0.000,C 90.000,E1 353.742} C_DIS
LIN {X -0.059,Y -191.071,Z 1451.933,A 0.000,B 0.000,C 90.000,E1 347.993} C_DIS
LIN {X -0.016,Y -194.000,Z 1451.897,A 0.000,B 0.000,C 90.000,E1 341.402} C_DIS
LIN {X 0.038,Y -197.610,Z 1451.869,A 0.000,B 0.000,C 90.000,E1 336.485} C_DIS
LIN {X 0.030,Y -201.764,Z 1451.847,A 0.000,B 0.000,C 90.000,E1 332.436} C_DIS
LIN {X 0.088,Y -207.099,Z 1451.825,A 0.000,B 0.000,C 90.000,E1 328.408} C_DIS
LIN {X -0.020,Y -212.316,Z 1451.807,A 0.000,B 0.000,C 90.000,E1 325.261} C_DIS
LIN {X 0.024,Y -218.467,Z 1451.790,A 0.000,B 0.000,C 90.000,E1 322.110} C_DIS
LIN {X 0.018,Y -225.538,Z 1451.772,A 0.000,B 0.000,C 90.000,E1 319.013} C_DIS
LIN {X -0.012,Y -233.599,Z 1451.755,A 0.000,B 0.000,C 90.000,E1 315.972} C_DIS
LIN {X 0.003,Y -242.533,Z 1451.739,A 0.000,B 0.000,C 90.000,E1 312.975} C_DIS
LIN {X 0.113,Y -252.641,Z 1451.722,A 0.000,B 0.000,C 90.000,E1 310.011} C_DIS
LIN {X 0.007,Y -263.923,Z 1451.706,A 0.000,B 0.000,C 90.000,E1 307.156} C_DIS
LIN {X 0.002,Y -271.652,Z 1451.697,A 0.000,B 0.000,C 90.000,E1 305.391} C_DIS
LIN {X 0.064,Y -281.981,Z 1451.685,A 0.000,B 0.000,C 90.000,E1 303.293} C_DIS
LIN {X 0.030,Y -291.641,Z 1451.676,A 0.000,B 0.000,C 90.000,E1 301.592} C_DIS
LIN {X 0.001,Y -302.332,Z 1451.666,A 0.000,B 0.000,C 90.000,E1 299.922} C_DIS
LIN {X -0.056,Y -311.894,Z 1451.659,A 0.000,B 0.000,C 90.000,E1 298.615} C_DIS
LIN {X -0.001,Y -322.398,Z 1451.652,A 0.000,B 0.000,C 90.000,E1 297.334} C_DIS
LIN {X 0.074,Y -335.832,Z 1451.644,A 0.000,B 0.000,C 90.000,E1 295.848} C_DIS
LIN {X 0.007,Y -349.588,Z 1451.636,A 0.000,B 0.000,C 90.000,E1 294.463} C_DIS
LIN {X 0.078,Y -363.180,Z 1451.628,A 0.000,B 0.000,C 90.000,E1 293.078} C_DIS
LIN {X -0.010,Y -373.483,Z 1451.622,A 0.000,B 0.000,C 90.000,E1 292.025} C_DIS
LIN {X 0.144,Y -386.485,Z 1451.615,A 0.000,B 0.000,C 90.000,E1 290.610} C_DIS
LIN {X 0.043,Y -396.641,Z 1451.608,A 0.000,B 0.000,C 90.000,E1 289.504} C_DIS
LIN {X -0.156,Y -409.086,Z 1451.601,A 0.000,B 0.000,C 90.000,E1 288.127} C_DIS
LIN {X 0.031,Y -416.213,Z 1451.596,A 0.000,B 0.000,C 90.000,E1 287.275} C_DIS
LIN {X 0.118,Y -422.905,Z 1451.591,A 0.000,B 0.000,C 90.000,E1 286.441} C_DIS
LIN {X -0.136,Y -428.895,Z 1451.587,A 0.000,B 0.000,C 90.000,E1 285.662} C_DIS
LIN {X -0.218,Y -432.396,Z 1451.584,A 0.000,B 0.000,C 90.000,E1 285.134} C_DIS
LIN {X 0.021,Y -436.816,Z 1451.579,A 0.000,B 0.000,C 90.000,E1 284.300} C_DIS
LIN {X -0.226,Y -440.448,Z 1451.575,A 0.000,B 0.000,C 90.000,E1 283.536} C_DIS
